IF Mach_Control.U.TJ_iMode=1 OR AV THEN//在自动状态下
CASE 	Sticker_Step2 OF
		0://判断备胶是否完成，贴胶冶具夹爪张开
				IF Mach_Control.TJ_b.StickPermit THEN//贴胶允许
						Sticker_Step2:=100;
				END_IF
		100:
				Mach_Control.TJ_b.StickPermit:=FALSE;//贴胶允许
				Mach_Control.TJ_b.StickFinish:=FALSE;//贴胶完成			
				Sticker_Step2:=200;
		200:
				IF NOT Sticker_SinStepMode THEN		
						IF 	Mach_Control.TJ_b.StickerStandbyDone  THEN//备胶完成,	
								Sticker_Step2:=250;						
						END_IF
				END_IF
		250: 
			IF arrCyCtrl[arrCyNo.ElectValveName.PastesGlueVacuum].Io.DOStatus1  
			AND arrCyCtrl[arrCyNo.ElectValveName.PastesGlueVacuum].Io.DIOnSwitch THEN
				Sticker_Step2:=300;
			ELSE
				Mach_Control.TJ_b.StickerStandbyDone:=FALSE;
				Mach_Control.TJ_b.Error[11]:=TRUE;//叠台贴胶头贴胶时无贴胶报警
				Sticker_Step2:=200;	
			END_IF
		
		300:
		arrAxisCtrl[AxiseNo.AxisName.GluingRetracting].Cmd.fOverride:=100;
				IF Mach_Control.TJ_b.Sticking_L THEN//左短边贴胶
					Sticker_Step2:=400;		
				ELSIF  Mach_Control.TJ_b.Sticking_R THEN//右短边贴胶
					Sticker_Step2:=450;		
				ELSIF Mach_Control.TJ_b.Sticking_Lg THEN//非极耳侧长边贴胶
					Sticker_Step2:=500;	
				ELSIF Mach_Control.TJ_b.Sticking_Lg2  THEN//极耳侧长边贴胶
					Sticker_Step2:=550;				
				END_IF	
		400://贴胶头移动左短边贴胶位
				IF NOT Sticker_SinStepMode THEN		
							IF GluingRetractingagree 
									AND  arrAxisCtrl[AxiseNo.AxisName.GluingRetracting].Status.Homed 
									AND arrAxisCtrl[AxiseNo.AxisName.GluingRetracting].Status.NoMoving 
									AND arrCyCtrl[arrCyNo.CylinderName.GlueClampsCy].Status.OFFState THEN
									IF arrAxisCtrl[AxiseNo.AxisName.GluingRetracting].Cmd.arrbRealPoint[2] THEN
											Mach_Control.TJ_b.Sticking_L:=FALSE;//左短边贴胶
											arrAxisCtrl[AxiseNo.AxisName.GluingRetracting].Cmd.iGoSetPos:=0;
											arrCyCtrl[arrCyNo.ElectValveName.PastesGlueVacuum].Cmd.bOFF:=TRUE;//备胶贴胶头真空关
											IF Mach_Control.TJ_b.SinStepMode THEN//贴胶单眇模式
													Sticker_SinStepMode:=TRUE;
											ELSE
													Sticker_SinStepMode:=FALSE;
											END_IF																						
											Sticker_Step2:=600;
									ELSE
											arrAxisCtrl[AxiseNo.AxisName.GluingRetracting].Cmd.iGoSetPos:=2;//贴胶头前进到贴胶位
									END_IF
										
							END_IF
							IF LREAL_TO_REAL(arrAxisCtrl[AxiseNo.AxisName.GluingRetracting].Status.fActPos) >= (arrAxisPar[AxiseNo.AxisName.GluingRetracting].arrTargetPoint[2]-30) THEN
									arrAxisCtrl[AxiseNo.AxisName.GluingRetracting].Cmd.fOverride:=5;
							END_IF
				END_IF
		450://贴胶头移动右短边贴胶位
				IF NOT Sticker_SinStepMode THEN		
						IF GluingRetractingagree 
						AND arrAxisCtrl[AxiseNo.AxisName.GluingRetracting].Status.Homed 
						AND arrAxisCtrl[AxiseNo.AxisName.GluingRetracting].Status.NoMoving 
						AND arrCyCtrl[arrCyNo.CylinderName.GlueClampsCy].Status.OFFState THEN
								IF arrAxisCtrl[AxiseNo.AxisName.GluingRetracting].Cmd.arrbRealPoint[3] THEN
										Mach_Control.TJ_b.Sticking_R:=FALSE;//左短边贴胶
										arrAxisCtrl[AxiseNo.AxisName.GluingRetracting].Cmd.iGoSetPos:=0;							
										arrCyCtrl[arrCyNo.ElectValveName.PastesGlueVacuum].Cmd.bOFF:=TRUE;//备胶贴胶头真空关
										IF Mach_Control.TJ_b.SinStepMode THEN//贴胶单眇模式
												Sticker_SinStepMode:=TRUE;
										ELSE
												Sticker_SinStepMode:=FALSE;
										END_IF																						
										Sticker_Step2:=600;
								ELSE
										arrAxisCtrl[AxiseNo.AxisName.GluingRetracting].Cmd.iGoSetPos:=3;//贴胶头前进到贴胶位
								END_IF	
						END_IF	
							IF LREAL_TO_REAL(arrAxisCtrl[AxiseNo.AxisName.GluingRetracting].Status.fActPos) >= (arrAxisPar[AxiseNo.AxisName.GluingRetracting].arrTargetPoint[3]-30) THEN
									arrAxisCtrl[AxiseNo.AxisName.GluingRetracting].Cmd.fOverride:=5;
							END_IF							
				END_IF
		500://非极耳侧长边贴胶
				IF NOT Sticker_SinStepMode THEN		
					IF GluingRetractingagree 
					AND arrAxisCtrl[AxiseNo.AxisName.GluingRetracting].Status.Homed 
					AND arrAxisCtrl[AxiseNo.AxisName.GluingRetracting].Status.NoMoving 
					AND arrCyCtrl[arrCyNo.CylinderName.GlueClampsCy].Status.OFFState THEN
						IF arrAxisCtrl[AxiseNo.AxisName.GluingRetracting].Cmd.arrbRealPoint[4] THEN
								Mach_Control.TJ_b.Sticking_Lg:=FALSE;//非极耳侧长边贴胶
								arrAxisCtrl[AxiseNo.AxisName.GluingRetracting].Cmd.iGoSetPos:=0;							
								arrCyCtrl[arrCyNo.ElectValveName.PastesGlueVacuum].Cmd.bOFF:=TRUE;//备胶贴胶头真空关
								IF Mach_Control.TJ_b.SinStepMode THEN//贴胶单眇模式
										Sticker_SinStepMode:=TRUE;
								ELSE
										Sticker_SinStepMode:=FALSE;
								END_IF																						
								Sticker_Step2:=600;
						ELSE
								arrAxisCtrl[AxiseNo.AxisName.GluingRetracting].Cmd.iGoSetPos:=4;//贴胶头前进到贴长边位
						END_IF		
					END_IF	
							IF LREAL_TO_REAL(arrAxisCtrl[AxiseNo.AxisName.GluingRetracting].Status.fActPos) >= (arrAxisPar[AxiseNo.AxisName.GluingRetracting].arrTargetPoint[4]-30) THEN
									arrAxisCtrl[AxiseNo.AxisName.GluingRetracting].Cmd.fOverride:=5;
							END_IF
				END_IF
	
			550://极耳侧长边贴胶
				IF NOT Sticker_SinStepMode THEN		
					IF GluingRetractingagree 
					AND arrAxisCtrl[AxiseNo.AxisName.GluingRetracting].Status.Homed 
					AND arrAxisCtrl[AxiseNo.AxisName.GluingRetracting].Status.NoMoving 
					AND arrCyCtrl[arrCyNo.CylinderName.GlueClampsCy].Status.OFFState THEN
						IF arrAxisCtrl[AxiseNo.AxisName.GluingRetracting].Cmd.arrbRealPoint[5] THEN
								Mach_Control.TJ_b.Sticking_Lg2:=FALSE;//极耳侧长边贴胶
								arrAxisCtrl[AxiseNo.AxisName.GluingRetracting].Cmd.iGoSetPos:=0;							
								arrCyCtrl[arrCyNo.ElectValveName.PastesGlueVacuum].Cmd.bOFF:=TRUE;//备胶贴胶头真空关
								IF Mach_Control.TJ_b.SinStepMode THEN//贴胶单眇模式
										Sticker_SinStepMode:=TRUE;
								ELSE
										Sticker_SinStepMode:=FALSE;
								END_IF																						
								Sticker_Step2:=600;
						ELSE
								arrAxisCtrl[AxiseNo.AxisName.GluingRetracting].Cmd.iGoSetPos:=5;//贴胶头前进到贴长边位
						END_IF		
					END_IF	
							IF LREAL_TO_REAL(arrAxisCtrl[AxiseNo.AxisName.GluingRetracting].Status.fActPos) >= (arrAxisPar[AxiseNo.AxisName.GluingRetracting].arrTargetPoint[5]-30) THEN
									arrAxisCtrl[AxiseNo.AxisName.GluingRetracting].Cmd.fOverride:=5;
							END_IF
				END_IF
			
		600:	
				IF NOT Sticker_SinStepMode THEN	
						TON_Sticker[4].IN:=FALSE;
						arrCyCtrl[arrCyNo.CylinderName.GlueClampsCy].Cmd.bON:=TRUE;//贴胶夹爪气缸夹紧
						IF arrCyCtrl[arrCyNo.CylinderName.GlueClampsCy].Status.ONState AND NOT arrCyCtrl[arrCyNo.CylinderName.GlueClampsCy].Status.Error1 THEN
								IF Mach_Control.TJ_b.SinStepMode THEN//贴胶单眇模式
									Sticker_SinStepMode:=TRUE;
								ELSE
									Sticker_SinStepMode:=FALSE;
								END_IF		
						TON_Sticker[4].IN:=TRUE;
							IF TON_Sticker[4].Q THEN
								Sticker_Step2:=700;	
								TON_Sticker[4].IN:=FALSE;
							END_IF		
						END_IF
				END_IF
		700:				
				IF NOT Sticker_SinStepMode THEN	
						arrCyCtrl[arrCyNo.CylinderName.GlueClampsCy].Cmd.bOFF:=TRUE;//贴胶夹爪气缸松开
						IF arrCyCtrl[arrCyNo.CylinderName.GlueClampsCy].Status.OFFState AND NOT arrCyCtrl[arrCyNo.CylinderName.GlueClampsCy].Status.Error2 THEN
								IF Mach_Control.TJ_b.SinStepMode THEN//贴胶单眇模式
										Sticker_SinStepMode:=TRUE;
								ELSE
										Sticker_SinStepMode:=FALSE;
								END_IF	
								arrAxisCtrl[AxiseNo.AxisName.GluingRetracting].Cmd.fOverride:=100;		
								Sticker_Step2:=800;
						END_IF
				END_IF
		800:
					IF NOT Sticker_SinStepMode THEN		
							IF GluingRetractingagree AND  arrAxisCtrl[AxiseNo.AxisName.GluingRetracting].Status.Homed AND arrAxisCtrl[AxiseNo.AxisName.GluingRetracting].Status.NoMoving THEN
									IF arrAxisCtrl[AxiseNo.AxisName.GluingRetracting].Cmd.arrbRealPoint[1] THEN
											arrAxisCtrl[AxiseNo.AxisName.GluingRetracting].Cmd.iGoSetPos:=0;
											Mach_Control.TJ_b.StickerStandbyDone:=FALSE;//复位备胶完成
											Mach_Control.TJ_b.StickFinish :=TRUE;//贴胶完成	
											Mach_Control.TJ_b.StickPermit:=false;//贴胶允许复位	
											IF Mach_Control.TJ_b.SinStepMode THEN//贴胶单眇模式
													Sticker_SinStepMode:=TRUE;
											ELSE
													Sticker_SinStepMode:=FALSE;
											END_IF																						
											Sticker_Step2:=900;
									ELSE
										arrAxisCtrl[AxiseNo.AxisName.GluingRetracting].Cmd.iGoSetPos:=1;//贴胶头前进到初始位
									END_IF
							END_IF	
					END_IF
			900:
					Sticker_Step2:=0;	
END_CASE
END_IF


CASE Sticker_Step0 OF
			1100://贴胶完成，允许下电芯，等待下电芯夹紧完成				
				IF Mach_Control.TJ_b.StickerOffloadingDone THEN
					Mach_Control.TJ_b.StickerFlag:=FALSE;
					Mach_Control.TJ_b.StickerOffloadingDone:=FALSE;						
					Sticker_Step0:=1200;
				END_IF
END_CASE


IF Sticker_Step0=4600 THEN
	Mach_Control.TJ_b.Stick_Judge:=TRUE;
ELSIF Sticker_Step0=2100 AND Sticker_Step0=2600 AND Sticker_Step0=3100 AND Sticker_Step0=3600 THEN
	Mach_Control.TJ_b.Stick_Judge:=FALSE;
END_IF
END_ACTION

ACTION _02BlueGlue_Auto:

(*
//蓝胶检测自动
DT_BlueGlue(
	Enable:=Mach_Control.U.DT_iMode=1 , //启动条件
	BlueSenser:=Mach_Control.se.BlueGluetsensor , //蓝胶检测信号
	An_Quantited:=Mach_Control.An_b.An_Quantited, //正极已叠极片数
	An_QuantitSet:=Par.stDT_date.An_Quantity , //正极设置极片数
	Ca_Quantited:=Mach_Control.Ca_b.Ca_Quantited, //负极已叠极片数
	Ca_QuantitSet:=Par.stDT_date.Ca_Quantity ,//负极设定极片数 
	Distance:=Par.stDT_date.Distance , //蓝胶检测到压刀的距离
	BluWidth:=Par.stDT_date.BluWidth , //蓝胶宽度
	Width:=Par.stDT_date.Width , //压刀外边宽
	BluGlueNG:=Mach_Control.DT_b.BluGlueNG );//电当蓝胶NG输出
	
	

//蓝胶标记
P2M_BlueFlag(
	Bnt_Blueflag:=Mach_Control.DT_b.stBnt_Blueflag , //蓝胶标记启动信号
	FlagDone:=P2M_BlueFlag.FlagDone , //蓝胶标记完成
	AixsoActPos:=arrAxis[AxiseNo.AxisName.SEPTAunwinding].NcToPlc.ActPos , //放卷轴当前位置
	Diameter:=Mach_Control.DT_b.fWindDiameter , //放卷轴当前卷径
	SetLenght:=Par.stDT_date.stSetLenght,//接带点到叠台的距离 3800
	fYDLength :=par.stDT_date.Width,
	rBnt_BlueflagCaNum :=Mach_Control.Ca_b.Ca_Quantited   , //叠台压刀外边宽
	FlagPoisn=> , //蓝胶NG标记
	NumberPos:=stNumberPos,//前一片数据
	NumberPos1:=stNumberPos1,//当前片数据
	NumberPos2:=stNumberPos2,
	rBnt_BlueflagNum :=DT_Ca_Quantited ,
	rBnt_Blueflaging:=Bnt_Blueflaging );//
	P2M_BlueFlag.FlagPoisn;	
	//
BulebntR_TRIG(CLK:=Mach_Control.DT_b.stBnt_Blueflag AND Mach_Control.DT_b.DT_Blue_TF   (*OR Mach_Control.btn.PoleInflationbtn*) , Q=> );
IF BulebntR_TRIG.Q THEN
	Bnt_Blueflaging:=TRUE;
	IF  (Par.stDT_date.An_Quantity+Par.stDT_date.Ca_Quantity-Mach_Control.An_b.An_Quantited-Mach_Control.Ca_b.Ca_Quantited)>=40 THEN
		Blueflaging:=TRUE;
	END_IF
END_IF	
*)
END_ACTION

ACTION _02Sticker_Auto:

TON_Sticker[0](PT:=T#0.2S);//拉胶气缸取胶延时
TON_Sticker[1](PT:=T#10S);//扫码超时报警延时
TON_Sticker[2](PT:=T#0.2S);//扫码超时报警延时
TON_Sticker[3](PT:=T#300MS);//扫码超时报警延时

IF Mach_Control.U.TJ_iMode<>1  THEN
				//一键备二维码胶
				rStickerStandbyCode_btn(CLK:=Mach_Control.btn.codeGluebtn , Q=> );
				fStickerStandbyCode_btn(CLK:=Mach_Control.btn.codeGluebtn , Q=> );
				IF rStickerStandbyCode_btn.Q THEN
					Mach_Control.TJ_b.StickerStandbyDone :=FALSE;
				END_IF
				IF fStickerStandbyCode_btn.Q THEN
					StandbyBule_Start:=FALSE;
					StandbyCode_Start:=TRUE;
				END_IF
				//一键备蓝胶
				rStickerStandbyBule_btn(CLK:=Mach_Control.btn.BlueGluebtn , Q=> );
				fStickerStandbyBule_btn(CLK:=Mach_Control.btn.BlueGluebtn , Q=> );
				IF rStickerStandbyBule_btn.Q THEN
					Mach_Control.TJ_b.StickerStandbyDone :=FALSE;
				END_IF
				IF fStickerStandbyBule_btn.Q THEN
					StandbyCode_Start:=FALSE;
					StandbyBule_Start:=TRUE;
				END_IF
END_IF

IF  StandbyBule_Start  THEN		
		Mach_Control.TJ_b.StickerStandbyBule:=FALSE;
END_IF

(*
//判断需要备什么胶,当设置的贴胶屏蔽时，置位已贴胶标记
IF Mach_Control.U.TJ_iMode=1 OR AV   THEN
			IF  NOT Mach_Control.TJ_b.StickerDoneNo[1]  AND NOT Mach_Control.TJ_b.Stickersetting[0]  THEN
				Mach_Control.TJ_b.StickerStandbyBule:=FALSE;//蓝胶备胶
				Mach_Control.TJ_b.StickerStandbyCode:=TRUE;//二维码备胶
				StandbyCode_Start:=FALSE;
				StandbyBule_Start:=FALSE;
			ELSIF (NOT Mach_Control.TJ_b.StickerDoneNo[2]  AND NOT Mach_Control.TJ_b.Stickersetting[1]) OR 
					(NOT Mach_Control.TJ_b.StickerDoneNo[3]  AND NOT Mach_Control.TJ_b.Stickersetting[2]) OR 
					(NOT Mach_Control.TJ_b.StickerDoneNo[4]  AND NOT Mach_Control.TJ_b.Stickersetting[3]) OR 
					(NOT Mach_Control.TJ_b.StickerDoneNo[5]  AND NOT Mach_Control.TJ_b.Stickersetting[4]) OR 
					(NOT Mach_Control.TJ_b.StickerDoneNo[6]  AND NOT Mach_Control.TJ_b.Stickersetting[5]) OR 
					(NOT Mach_Control.TJ_b.StickerDoneNo[7]  AND NOT Mach_Control.TJ_b.Stickersetting[6]) THEN
				Mach_Control.TJ_b.StickerStandbyBule:=TRUE;//蓝胶备胶
				Mach_Control.TJ_b.StickerStandbyCode:=FALSE;//二维码备胶	
				StandbyCode_Start:=FALSE;
				StandbyBule_Start:=FALSE;		
			END_IF
END_IF
*)


GluingUpDownPoint1:=ABS(arrAxisPar[AxiseNo.AxisName.GluingUpDown].arrTargetPoint[1]-arrAxisPar[AxiseNo.AxisName.GluingUpDown].arrTargetPoint[2]);
GluingUpDownPoint3:=ABS(GluingUpDownPoint2-arrAxisPar[AxiseNo.AxisName.GluingUpDown].arrTargetPoint[1]);
IF GluingUpDownPoint3-GluingUpDownPoint1>=2 THEN
	GluingUpDownPoint4:=2;
ELSIF GluingUpDownPoint3-GluingUpDownPoint1<=-2 THEN
	GluingUpDownPoint4:=-2;
ELSE
	GluingUpDownPoint4:=GluingUpDownPoint3-GluingUpDownPoint1;
END_IF

rMarkesensorR_TRIG(CLK:=Mach_Control.se.Markesensor , Q=> );

IF (Mach_Control.U.TJ_iMode=1 OR StandbyCode_Start OR StandbyBule_Start OR AV) AND NOT TJ_Error THEN//在自动状态下
	
//贴胶备胶自动
	
CASE Sticker_Step1 OF
		0://判断贴胶备胶是否完成
				IF NOT Sticker_SinStepMode THEN
						IF NOT Mach_Control.TJ_b.StickerStandbyDone THEN//备胶没有完成，贴胶头前进后退轴在安全位
								IF Mach_Control.TJ_b.SinStepMode THEN//贴胶单眇模式
									Sticker_SinStepMode:=TRUE;
								ELSE
									Sticker_SinStepMode:=FALSE;
								END_IF
								Sticker_Step1:=10;					
						END_IF
				END_IF
		10://备二维码胶真空1、备蓝胶真空1	
				//arrCyCtrl[arrCyNo.ElectValveName.codeGlueVacuum1].Cmd.bON:=TRUE;//备二维码胶真空1						
				arrCyCtrl[arrCyNo.ElectValveName.BlueGlueVacuum1].Cmd.bON:=TRUE;//备蓝胶真空1					
				Sticker_Step1:=20;			
		20://贴胶台具气缸张开、贴胶头前进轴回初始位
				IF NOT Sticker_SinStepMode THEN
						IF(GluingRetractingagree OR  arrAxisCtrl[AxiseNo.AxisName.GluingRetracting].Cmd.arrbRealPoint[1])AND
							arrAxisCtrl[AxiseNo.AxisName.GluingRetracting].Status.Homed AND arrAxisCtrl[AxiseNo.AxisName.GluingRetracting].Status.NoMoving THEN
								IF arrAxisCtrl[AxiseNo.AxisName.GluingRetracting].Cmd.arrbRealPoint[1] THEN
										arrAxisCtrl[AxiseNo.AxisName.GluingRetracting].Cmd.iGoSetPos:=0;						
										IF Mach_Control.TJ_b.SinStepMode THEN//贴胶单眇模式
												Sticker_SinStepMode:=TRUE;
										ELSE
												Sticker_SinStepMode:=FALSE;
										END_IF
										Sticker_Step1:=30;
								ELSE
										arrAxisCtrl[AxiseNo.AxisName.GluingRetracting].Cmd.iGoSetPos:=1;//贴胶头前进到贴胶位
								END_IF
						END_IF
				END_IF					
	   30://贴胶压胶气缸伸出，备胶气缸伸出
				IF NOT Sticker_SinStepMode THEN  
						arrCyCtrl[arrCyNo.CylinderName.GluePressCy].Cmd.bON:=TRUE;//贴胶压胶气缸伸出
						arrCyCtrl[arrCyNo.CylinderName.CodeGluePressCy].Cmd.bON:=TRUE;//贴胶压二维码胶气缸伸出
						IF arrCyCtrl[arrCyNo.CylinderName.CodeGluePressCy].Io.DIOnSwitch THEN
								arrCyCtrl[arrCyNo.CylinderName.CodeStandbyGlueCy].Cmd.bON:=TRUE;//贴胶备二维码胶气缸伸出
						END_IF
						IF Mach_Control.TJ_b.SinStepMode THEN//贴胶单眇模式
								Sticker_SinStepMode:=TRUE;
						ELSE
								Sticker_SinStepMode:=FALSE;
						END_IF
						IF arrCyCtrl[arrCyNo.CylinderName.GluePressCy].Status.ONState AND arrCyCtrl[arrCyNo.CylinderName.CodeGluePressCy].Status.ONState THEN
								Sticker_Step1:=40;	
						END_IF
				END_IF
		40://判断贴蓝胶、二维码胶
				IF NOT Sticker_SinStepMode THEN
					//IF Mach_Control.TJ_b.StickerStandbyBule OR StandbyBule_Start THEN//备蓝胶请求
					IF Mach_Control.TJ_b.SinStepMode THEN//贴胶单眇模式
							Sticker_SinStepMode:=TRUE;
					ELSE
							Sticker_SinStepMode:=FALSE;
					END_IF								
					arrCyCtrl[arrCyNo.CylinderName.StandbyGlueCy].Cmd.bON:=TRUE;//备蓝胶气缸伸出
					IF 	arrCyCtrl[arrCyNo.CylinderName.StandbyGlueCy].Io.DIOnSwitch THEN
							Sticker_Step1:=200;
					END_IF
					//END_IF	
				END_IF			
		200:// 二维码胶、蓝胶切胶气缸伸出，拉胶气缸伸出，拉胶升降轴移至拉蓝胶起始位
				IF NOT Sticker_SinStepMode THEN			
						arrCyCtrl[arrCyNo.CylinderName.codeGlueCutCy].Cmd.bON:=TRUE;//贴胶切二维码胶气缸伸出
						arrCyCtrl[arrCyNo.CylinderName.GlueCutCy].Cmd.bON:=TRUE;//贴胶切胶气缸伸出
						arrCyCtrl[arrCyNo.CylinderName.PullGlueCy].Cmd.bON:=TRUE;//拉胶气缸伸出
						arrCyCtrl[arrCyNo.CylinderName.StandbyGlueCy].Cmd.bOFF:=TRUE;//备蓝胶气缸伸出
						IF  GluingUpDownagree AND arrAxisCtrl[AxiseNo.AxisName.GluingUpDown].Status.Homed AND arrAxisCtrl[AxiseNo.AxisName.GluingUpDown].Status.NoMoving THEN
								IF arrAxisCtrl[AxiseNo.AxisName.GluingUpDown].Cmd.arrbRealPoint[9] THEN
										arrAxisCtrl[AxiseNo.AxisName.GluingUpDown].Cmd.iGoSetPos:=0;
										IF Mach_Control.TJ_b.SinStepMode THEN//贴胶单眇模式
												Sticker_SinStepMode:=TRUE;
										ELSE
												Sticker_SinStepMode:=FALSE;
										END_IF
										Sticker_Step1:=205;	
								ELSE
										arrAxisCtrl[AxiseNo.AxisName.GluingUpDown].Cmd.iGoSetPos:=9;//拉胶升降轴至拉蓝胶起始位
								END_IF
						END_IF		
				END_IF
		205:
				IF NOT Sticker_SinStepMode THEN
						IF  GluingUpDownagree AND arrAxisCtrl[AxiseNo.AxisName.GluingUpDown].Status.Homed AND arrAxisCtrl[AxiseNo.AxisName.GluingUpDown].Status.NoMoving THEN
								IF arrAxisCtrl[AxiseNo.AxisName.GluingUpDown].Cmd.arrbRealPoint[3] THEN
										arrAxisCtrl[AxiseNo.AxisName.GluingUpDown].Cmd.iGoSetPos:=0;
										IF Mach_Control.TJ_b.SinStepMode THEN//贴胶单眇模式
												Sticker_SinStepMode:=TRUE;
										ELSE
												Sticker_SinStepMode:=FALSE;
										END_IF
										Sticker_Step1:=210;	
								ELSE
										arrAxisCtrl[AxiseNo.AxisName.GluingUpDown].Cmd.iGoSetPos:=3;//拉胶升降轴至拉蓝胶起始位
								END_IF
						END_IF		
				END_IF
			210://拉胶升降气缸收回,取胶
				IF NOT Sticker_SinStepMode THEN			
						arrCyCtrl[arrCyNo.CylinderName.PullGlueCy].Cmd.bOFF:=TRUE;//拉胶气缸收回	
						arrCyCtrl[arrCyNo.CylinderName.GluePressCy].Cmd.bOFF:=TRUE;//贴胶压胶气缸伸出
						arrCyCtrl[arrCyNo.CylinderName.PullGluePoleCy].Cmd.bOFF:=TRUE;//拉胶抱紧气缸松开
						IF arrCyCtrl[arrCyNo.CylinderName.PullGlueCy].Io.DIOFFSwitch THEN
								IF NOT TON_Sticker[0].Q THEN
										TON_Sticker[0].IN:=TRUE;
								ELSE
										TON_Sticker[0].IN:=FALSE;
										IF Mach_Control.TJ_b.SinStepMode THEN//贴胶单眇模式
												Sticker_SinStepMode:=TRUE;
										ELSE
												Sticker_SinStepMode:=FALSE;
										END_IF
								Sticker_Step1:=220;
								END_IF
						END_IF	
				END_IF
		220://取胶滚胶位
				IF NOT Sticker_SinStepMode THEN			
						arrCyCtrl[arrCyNo.CylinderName.PullGluePoleCy].Cmd.bOFF:=TRUE;//拉胶抱紧气缸松开
						IF   arrAxisCtrl[AxiseNo.AxisName.GluingUpDown].Status.Homed AND arrAxisCtrl[AxiseNo.AxisName.GluingUpDown].Status.NoMoving THEN
								IF arrAxisCtrl[AxiseNo.AxisName.GluingUpDown].Cmd.arrbRealPoint[7] THEN
										arrAxisCtrl[AxiseNo.AxisName.GluingUpDown].Cmd.iGoSetPos:=0;
										IF Mach_Control.TJ_b.SinStepMode THEN//贴胶单眇模式
												Sticker_SinStepMode:=TRUE;
										ELSE
												Sticker_SinStepMode:=FALSE;
										END_IF
										Sticker_Step1:=221;	
								ELSE
										arrAxisCtrl[AxiseNo.AxisName.GluingUpDown].Cmd.iGoSetPos:=7;//拉胶升降轴取胶滚胶位
								END_IF
						END_IF
				END_IF	
		221://
				IF NOT Sticker_SinStepMode THEN
						IF NOT TON_Sticker[0].Q THEN
								arrCyCtrl[arrCyNo.ElectValveName.BlueGlueVacuum1].Cmd.bOFF:=TRUE;//备蓝胶真空1关
								arrCyCtrl[arrCyNo.ElectValveName.codeGlueVacuum2].Cmd.bOFF:=TRUE;//备二维码胶真空2关
								arrCyCtrl[arrCyNo.ElectValveName.PastesGlueVacuum].Cmd.bOFF:=TRUE;//备胶贴胶头真空关
								arrCyCtrl[arrCyNo.CylinderName.PullGluePoleCy].Cmd.bON:=TRUE;//拉胶抱紧气缸抱紧
								TON_Sticker[0].IN:=TRUE;
						ELSE
								TON_Sticker[0].IN:=FALSE;
								IF Mach_Control.TJ_b.SinStepMode THEN//贴胶单眇模式
										Sticker_SinStepMode:=TRUE;
								ELSE
										Sticker_SinStepMode:=FALSE;
								END_IF								
								Sticker_Step1:=230;	;	
						END_IF
				END_IF
		230://拉胶升降气缸伸出，拉胶升降气缸移动至拉蓝胶终点位
				IF NOT Sticker_SinStepMode THEN			
						arrCyCtrl[arrCyNo.CylinderName.codeGlueCutCy].Cmd.bON:=TRUE;//贴胶切二维码胶气缸伸出
						arrCyCtrl[arrCyNo.CylinderName.GlueCutCy].Cmd.bON:=TRUE;//贴胶切胶气缸伸出
						arrCyCtrl[arrCyNo.CylinderName.PullGlueCy].Cmd.bON:=TRUE;//拉胶气缸伸出
						arrCyCtrl[arrCyNo.CylinderName.PullGluePoleCy].Cmd.bON:=TRUE;//拉胶抱紧气缸抱紧
						IF  GluingUpDownagree AND arrAxisCtrl[AxiseNo.AxisName.GluingUpDown].Status.Homed AND arrAxisCtrl[AxiseNo.AxisName.GluingUpDown].Status.NoMoving THEN
								IF arrAxisCtrl[AxiseNo.AxisName.GluingUpDown].Cmd.arrbRealPoint[4] THEN
										arrAxisCtrl[AxiseNo.AxisName.GluingUpDown].Cmd.iGoSetPos:=0;
										IF Mach_Control.TJ_b.SinStepMode THEN//贴胶单眇模式
												Sticker_SinStepMode:=TRUE;
										ELSE
												Sticker_SinStepMode:=FALSE;
										END_IF
										Sticker_Step1:=240;	
								ELSE
										arrAxisCtrl[AxiseNo.AxisName.GluingUpDown].Cmd.iGoSetPos:=4;//拉胶升降轴至拉蓝胶终点位
								END_IF
						END_IF
				END_IF					
		240://拉胶气缸收回
				IF NOT Sticker_SinStepMode THEN			
						arrCyCtrl[arrCyNo.CylinderName.PullGlueCy].Cmd.bOFF:=TRUE;//拉胶气缸收回		
						arrCyCtrl[arrCyNo.CylinderName.PullGluePoleCy].Cmd.bOFF:=TRUE;//拉胶抱紧气缸松开	
						arrCyCtrl[arrCyNo.ElectValveName.BlueGlueVacuum1].Cmd.bON:=TRUE;//备蓝胶真空1
						arrCyCtrl[arrCyNo.ElectValveName.BlueGlueVacuum2].Cmd.bON:=TRUE;//备蓝胶真空2	
						arrCyCtrl[arrCyNo.ElectValveName.codeGlueVacuum1].Cmd.bON:=TRUE;//备二维码胶真空1
						arrCyCtrl[arrCyNo.ElectValveName.codeGlueVacuum2].Cmd.bON:=TRUE;//备二维码胶真空2																			
						IF arrCyCtrl[arrCyNo.CylinderName.PullGlueCy].Status.OFFState THEN
								IF NOT TON_Sticker[0].Q THEN
										TON_Sticker[0].IN:=TRUE;
								ELSE
										TON_Sticker[0].IN:=FALSE;
										IF Mach_Control.TJ_b.SinStepMode THEN//贴胶单眇模式
												Sticker_SinStepMode:=TRUE;
										ELSE
												Sticker_SinStepMode:=FALSE;
										END_IF					
								Sticker_Step1:=250;
								END_IF
						END_IF	
				END_IF
		250:	//拉胶升降轴至切胶滚胶位	
				IF NOT Sticker_SinStepMode THEN			
						IF   arrAxisCtrl[AxiseNo.AxisName.GluingUpDown].Status.Homed AND arrAxisCtrl[AxiseNo.AxisName.GluingUpDown].Status.NoMoving THEN
								IF arrAxisCtrl[AxiseNo.AxisName.GluingUpDown].Cmd.arrbRealPoint[8] THEN
										arrAxisCtrl[AxiseNo.AxisName.GluingUpDown].Cmd.iGoSetPos:=0;
										IF Mach_Control.TJ_b.SinStepMode THEN//贴胶单眇模式
												Sticker_SinStepMode:=TRUE;
										ELSE
												Sticker_SinStepMode:=FALSE;
										END_IF
										Sticker_Step1:=255;	
								ELSE
										arrAxisCtrl[AxiseNo.AxisName.GluingUpDown].Cmd.iGoSetPos:=8;//拉胶升降轴至切胶滚胶位
								END_IF
						END_IF
				END_IF	
	
		255://20230205修改切胶动作
				arrCyCtrl[arrCyNo.CylinderName.GluePressCy].Cmd.bON:=TRUE;//贴胶压胶气缸伸出
				IF arrCyCtrl[arrCyNo.CylinderName.GluePressCy].Status.ONState THEN//贴胶压胶气缸伸出
						Sticker_Step1:=260;		
				END_IF
		
		260://切二维码胶气缸收回，切胶
				IF NOT Sticker_SinStepMode THEN	
						arrCyCtrl[arrCyNo.ElectValveName.PastesGlueVacuum].Cmd.bON:=TRUE;//备胶贴胶头真空		
						arrCyCtrl[arrCyNo.CylinderName.GlueCutCy].Cmd.bOFF:=TRUE;//切蓝胶气缸收回
						IF arrCyCtrl[arrCyNo.CylinderName.GlueCutCy].Status.OFFState THEN													
									IF Mach_Control.TJ_b.SinStepMode THEN//贴胶单眇模式
											Sticker_SinStepMode:=TRUE;
									ELSE
											Sticker_SinStepMode:=FALSE;
									END_IF															
									Sticker_Step1:=270;	
						END_IF	
				END_IF
		270://拉胶气缸伸出、切胶气缸伸出、拉胶升降轴回初始位
				IF NOT Sticker_SinStepMode THEN			
						arrCyCtrl[arrCyNo.CylinderName.codeGlueCutCy].Cmd.bON:=TRUE;//贴胶切二维码胶气缸伸出
						arrCyCtrl[arrCyNo.CylinderName.GlueCutCy].Cmd.bON:=TRUE;//贴胶切胶气缸伸出
						arrCyCtrl[arrCyNo.CylinderName.PullGlueCy].Cmd.bON:=TRUE;//拉胶气缸伸出
						arrCyCtrl[arrCyNo.ElectValveName.BlueGlueVacuum2].Cmd.bON:=FALSE;//备蓝胶真空2	
						arrCyCtrl[arrCyNo.ElectValveName.codeGlueVacuum2].Cmd.bON:=FALSE;//备二维码胶真空2
						arrCyCtrl[arrCyNo.ElectValveName.BlueGlueVacuum2].Cmd.bOFF:=TRUE;//备蓝胶真空2	
						arrCyCtrl[arrCyNo.ElectValveName.codeGlueVacuum2].Cmd.bOFF:=TRUE;//备二维码胶真空2								
						IF  GluingUpDownagree AND arrAxisCtrl[AxiseNo.AxisName.GluingUpDown].Status.Homed AND arrAxisCtrl[AxiseNo.AxisName.GluingUpDown].Status.NoMoving THEN
								IF arrAxisCtrl[AxiseNo.AxisName.GluingUpDown].Cmd.arrbRealPoint[9] THEN
										arrAxisCtrl[AxiseNo.AxisName.GluingUpDown].Cmd.iGoSetPos:=0;
										IF Mach_Control.TJ_b.SinStepMode THEN//贴胶单眇模式
												Sticker_SinStepMode:=TRUE;
										ELSE
												Sticker_SinStepMode:=FALSE;
										END_IF
										Mach_Control.TJ_b.StickerStandbyDone:=TRUE;
										StandbyBule_Start:=FALSE;
										arrCyCtrl[arrCyNo.CylinderName.StandbyGlueCy].Cmd.bON:=TRUE;//备蓝胶气缸伸出		
										Sticker_Step1:=0;	
								ELSE
										arrAxisCtrl[AxiseNo.AxisName.GluingUpDown].Cmd.iGoSetPos:=9;//拉胶升降轴至拉蓝胶起始位
								END_IF
						END_IF		
				END_IF						
END_CASE
END_IF


IF Mach_Control.TJ_b.Error[5] AND Sticker_Step1>=260 AND Sticker_Step1<=270 THEN
	Sticker_Step1:=0;
	Mach_Control.TJ_b.StickerStandbyDone:=FALSE;
END_IF
END_ACTION

ACTION _02Sticker_AutoSbu1_Scan:
(*
Scan_TON[1](PT:=T#3MS);
Scan_TON[2](PT:=T#3MS);
Scan_TON[3](PT:=T#3MS);
Scan_TON[4](PT:=T#100MS);


//二维码胶扫码		
	CASE Stick_Step0 OF
		10:
			Scan_TON[1].IN:=FALSE;
			Scan_TON[2].IN:=FALSE;
			Scan_TON[3].IN:=FALSE;
			Stick_Step0:=20;
			
		20:
			fbinit_tcp:=TRUE;
			Scan_TON[1].IN:=TRUE;
			IF Scan_TON[1].Q THEN
				fbinit_tcp:=FALSE;
				Scan_TON[1].IN:=FALSE;
				Stick_Step0:=30;
			END_IF

		30:
			fbComOpen:=TRUE;
			Scan_TON[2].IN:=TRUE;
			IF Scan_TON[2].Q THEN
				fbComOpen:=FALSE;
				Scan_TON[2].IN:=FALSE;
				Stick_Step0:=40;
			END_IF

		40:
			IF bCS_CodeTcp.bComOpenDone THEN
				Stick_Step0:=50;
			END_IF
		
		50:
			bCS_CodeTcp.bLON:=TRUE;
			Scan_TON[3].IN:=TRUE;
			IF Scan_TON[3].Q THEN
				bCS_CodeTcp.bLON:=FALSE;
				Scan_TON[3].IN:=FALSE;
				Stick_Step0:=60;
			END_IF
		60:
			Scan_TON[4].IN:=TRUE;
			IF 	Scan_TON[4].Q THEN
				Stick_Step0:=70;
				Scan_TON[4].IN:=FALSE;
			END_IF

		70:
			IF  bCS_CodeTcp.Code_State=1  THEN
				Mach_Control.TJ_b.strCode:=bCS_CodeTcp.strCode;
				Mach_Control.TJ_b.Scan_gross:=bCS_CodeTcp.Code_State;
				Stick_Step0:=80;
				Mach_Control.TJ_b.ScanStarte:=FALSE;
				
			 ELSIF bCS_CodeTcp.Code_State=2 THEN
				 Mach_Control.TJ_b.Scan_gross:=bCS_CodeTcp.Code_State;
				 Stick_Step0:=80;
				 Mach_Control.TJ_b.ScanStarte:=FALSE;
			 ELSIF bCS_CodeTcp.bCodeConError OR Mach_Control.TJ_b.Error[0] THEN
				Stick_Step0:=6666;
				Mach_Control.TJ_b.ScanStarte:=FALSE;
			END_IF

	END_CASE

(*IF Mach_Control.TJ_b.ScanOK AND NOT   Mach_Control.TJ_b.ScanNG THEN
					Mach_Control.TJ_b.ScanStatus[0]:=TRUE;//扫码位的胶琮扫码OK
					Mach_Control.TJ_b.ScanStarte:=FALSE;//二维码扫码启动	
					TON_Sticker[1].IN:=FALSE;
					Stick_Step0:=6666;
				ELSIF NOT Mach_Control.TJ_b.ScanOK AND Mach_Control.TJ_b.ScanNG  THEN
					Mach_Control.TJ_b.ScanStatus[0]:=FALSE;//扫码位的胶琮扫码NG
					Mach_Control.TJ_b.ScanStarte:=FALSE;//二维码扫码启动	
					TON_Sticker[1].IN:=FALSE;	
					Stick_Step0:=6666;	
				ELSE
						IF NOT TON_Sticker[1].Q THEN
							TON_Sticker[1].IN:=TRUE;
						ELSE
							TON_Sticker[1].IN:=FALSE;
							Mach_Control.TJ_b.Error[0]:=TRUE;//扫码超时报警
							Mach_Control.TJ_b.ScanStarte:=FALSE;//二维码扫码启动	
							Stick_Step0:=9999;	
						END_IF
				END_IF*)

	
	
		
			
					
(*
上升沿触发 fbComOpen,  bComOpenDone连接完成；
触发fbLON拍照；
*)
bCS_CodeTcp(
	bLON:=bCS_CodeTcp.bLON,                           	// 扫码触发
	sRemoteHost:=Par.Code.sRemoteHost	,					//后段扫码枪；sRemoteHost:='192.168.10.25'
	bComOpen:=fbComOpen,           //扫码Tcp 连接，上升沿；
	binit_tcp:=fbinit_tcp,					//初始化功能块，上升沿；
	bComOpenDone=>, 			 //扫码Tcp 打开OK
    bCodeConError =>Mach_Control.TJ_b.Error[0],            	//扫码通讯故障
	bDone=>,                        	 //扫码完成
    bCodeError=>Mach_Control.TJ_b.Error[0],                  //扫码故障	
    strCode =>,                      //条码结果
	Code_State=>,					//扫码结果 1：OK  2：NG
);

bCS_CodeTcp.bDone;//这个需外部复位；
bCS_CodeTcp.strCode;
bCS_CodeTcp.Code_State;
bCS_CodeTcp.bComOpenDone;

*)
END_ACTION

ACTION _02Sticker_AutoSbu2_NG:

//贴胶踢废胶程序
		CASE 	Stick_Step2  OF 
		100://踢废胶
					arrCyCtrl[arrCyNo.CylinderName.GlueNGCy].Cmd.bON:=TRUE;//踢废胶升降气缸伸出
					IF 	 arrCyCtrl[arrCyNo.CylinderName.GlueNGCy].Io.DIOnSwitch THEN
						IF arrAxisCtrl[AxiseNo.AxisName.GluingRetracting].Status.Homed AND arrAxisCtrl[AxiseNo.AxisName.GluingRetracting].Status.NoMoving THEN
							IF arrAxisCtrl[AxiseNo.AxisName.GluingRetracting].Cmd.arrbRealPoint[6] THEN
								arrAxisCtrl[AxiseNo.AxisName.GluingRetracting].Cmd.iGoSetPos:=0;
								Mach_Control.TJ_b.StickerStandbyDone:=FALSE;//复位备胶完成
								IF Mach_Control.TJ_b.SinStepMode THEN//贴胶单眇模式
									Sticker_SinStepMode:=TRUE;
								ELSE
									Sticker_SinStepMode:=FALSE;
								END_IF																						
								Stick_Step2:=200;
							ELSE
								arrAxisCtrl[AxiseNo.AxisName.GluingRetracting].Cmd.iGoSetPos:=6;//踢废胶位
							END_IF
						END_IF	
					END_IF	
		120://贴胶冶具夹爪夹紧
					IF NOT Sticker_SinStepMode THEN		
						arrCyCtrl[arrCyNo.CylinderName.PullGlueModelCy].Cmd.bON:=TRUE;//贴胶冶具夹爪夹紧
						IF arrCyCtrl[arrCyNo.CylinderName.PullGlueModelCy].Io.DIOnSwitch THEN
							IF Mach_Control.TJ_b.SinStepMode THEN//贴胶单眇模式
								Sticker_SinStepMode:=TRUE;
							ELSE
								Sticker_SinStepMode:=FALSE;
							END_IF								
							Stick_Step2:=130;
						END_IF
					END_IF	
		130://贴胶夹爪张开，贴胶尖退回到初始位
					IF NOT Sticker_SinStepMode THEN		
							arrCyCtrl[arrCyNo.CylinderName.PullGlueModelCy].Cmd.bOFF:=TRUE;//贴胶冶具夹爪张开
							IF 	Mach_Control.TJ_b.StickerStandbyDone THEN
								IF arrCyCtrl[arrCyNo.CylinderName.PullGlueModelCy].Io.DIOFFSwitch AND arrAxisCtrl[AxiseNo.AxisName.GluingRetracting].Status.Homed AND arrAxisCtrl[AxiseNo.AxisName.GluingRetracting].Status.NoMoving THEN
									IF arrAxisCtrl[AxiseNo.AxisName.GluingRetracting].Cmd.arrbRealPoint[1] THEN
										arrAxisCtrl[AxiseNo.AxisName.GluingRetracting].Cmd.iGoSetPos:=0;
										IF Mach_Control.TJ_b.SinStepMode THEN//贴胶单眇模式
											Sticker_SinStepMode:=TRUE;
										ELSE
											Sticker_SinStepMode:=FALSE;
										END_IF																						
										Stick_Step2:=140;
									ELSE
										arrAxisCtrl[AxiseNo.AxisName.GluingRetracting].Cmd.iGoSetPos:=1;//贴胶头前进到备胶位
									END_IF
								END_IF						
						END_IF
					END_IF	
		140://踢废胶升降气缸纠回	
					arrCyCtrl[arrCyNo.CylinderName.GlueNGCy].Cmd.bOFF:=TRUE;//踢废胶升降气缸纠回
					IF 	arrCyCtrl[arrCyNo.CylinderName.GlueNGCy].Io	.DIOFFSwitch	THEN
						Stick_Step2:=6666;
					END_IF
		END_CASE
END_ACTION

ACTION _03Rectifydev_Auto:

//隔膜纠偏自动
IF Mach_Control.DT_b.RectifydevStarte OR Mach_Control.U.DT_iMode=1 OR (TailCurlStep3>=150 AND TailCurlStep3<=160  AND  Mach_Control.U.WJ_iMode=1 ) THEN
	 fbRectifyGM.Execute:=TRUE;
ELSE
	fbRectifyGM.Execute:=FALSE;
END_IF
//隔膜纠偏条件
(*
//fbRectifyGM.bRecEn:= arrAxis[AxiseNo.VirAxisName.VirGM].NcToPlc.SetVelo>=0.5 AND  ABS( arrAxis[AxiseNo.AxisName.SEPTATLine].NcToPlc.ActPos  )>=24 ;    //隔膜正向运动且隔膜包角OK位置 
fbRectifyGM.bRecEn:=((( 
                                    (LREAL_TO_REAL(arrAxisCtrl[AxiseNo.AxisName.SEPTATLine].Status.fActPos)>arrAxisPar[AxiseNo.AxisName.SEPTATLine].arrTargetPoint[1]+1    AND   
                                     LREAL_TO_REAL(arrAxisCtrl[AxiseNo.AxisName.SEPTATLine].Status.fActPos)<arrAxisPar[AxiseNo.AxisName.SEPTATLine].arrTargetPoint[1]+120) OR
                                    (LREAL_TO_REAL(arrAxisCtrl[AxiseNo.AxisName.SEPTATLine].Status.fActPos)<arrAxisPar[AxiseNo.AxisName.SEPTATLine].arrTargetPoint[2]-1    AND   
                                     LREAL_TO_REAL(arrAxisCtrl[AxiseNo.AxisName.SEPTATLine].Status.fActPos)>arrAxisPar[AxiseNo.AxisName.SEPTATLine].arrTargetPoint[2]-110) OR
									(TailCurlStep3>=1070 AND TailCurlStep3<=1080 AND  Mach_Control.U.WJ_iMode=1)                                                           OR 
                                    (TailCurlStep3>=150 AND TailCurlStep3<=160 AND  Mach_Control.U.WJ_iMode=1) AND Par.stDT_date.iRectifyMode=2))(* OR
									 (arrAxis[AxiseNo.VirAxisName.VirGM].NcToPlc.SetVelo>=5 AND  ABS( arrAxis[AxiseNo.AxisName.SEPTATLine].NcToPlc.ActPos  )>=24)  AND Par.stDT_date.iRectifyMode=1) *) OR Mach_Control.DT_b.RectifydevStarte) AND 
									 NOT Mach_Control.DT_b.RectifydevModel   ; //隔膜正向运动且隔膜包角OK位置 
*)

//纠偏条件		
(*							 
bRectifyRule[1]:=arrAxisCtrl[AxiseNo.AxisName.SEPTATLine].Status.fActPos>(arrAxisPar[AxiseNo.AxisName.SEPTATLine].arrTargetPoint[1]+5)    AND   
                                     arrAxisCtrl[AxiseNo.AxisName.SEPTATLine].Status.fSetPos<(arrAxisPar[AxiseNo.AxisName.SEPTATLine].arrTargetPoint[1]+Par.stDT_date.iRectifyAnPos);	//隔膜纠偏条件										 
									 
bRectifyRule[2]:=arrAxisCtrl[AxiseNo.AxisName.SEPTATLine].Status.fActPos<(arrAxisPar[AxiseNo.AxisName.SEPTATLine].arrTargetPoint[2]-5 )   AND   
                                     arrAxisCtrl[AxiseNo.AxisName.SEPTATLine].Status.fSetPos>(arrAxisPar[AxiseNo.AxisName.SEPTATLine].arrTargetPoint[2]-Par.stDT_date.iRectifyCaPos);
*)
								 
bRectifyRule[1]:=fbCamInGMDanserMove.iTableSel=2  AND   arrAxis[AxiseNo.AxisName.SEPTATLine].Status.Moving AND
                             arrAxisCtrl[AxiseNo.AxisName.SEPTATLine].Status.fSetPos<(arrAxisPar[AxiseNo.AxisName.SEPTATLine].arrTargetPoint[1]+Par.stDT_date.iRectifyAnPos);	//隔膜纠偏条件										 
									 
bRectifyRule[2]:=fbCamInGMDanserMove.iTableSel=1  AND   arrAxis[AxiseNo.AxisName.SEPTATLine].Status.Moving AND
                             arrAxisCtrl[AxiseNo.AxisName.SEPTATLine].Status.fSetPos>(arrAxisPar[AxiseNo.AxisName.SEPTATLine].arrTargetPoint[2]-Par.stDT_date.iRectifyCaPos);	
								 
bRectifyRule[3]:=TailCurlStep3>=1070 AND TailCurlStep3<=1080 AND  Mach_Control.U.WJ_iMode=1;		
bRectifyRule[4]:=TailCurlStep3>=150 AND TailCurlStep3<=160 AND  Mach_Control.U.WJ_iMode=1 AND Par.stDT_date.iRectifyMode=2;			
				 
fbRectifyGM.bRecEn:=NOT Mach_Control.DT_b.RectifydevModel AND( bRectifyRule[1] OR bRectifyRule[2] OR bRectifyRule[3] OR bRectifyRule[4] OR An_OverNGStep=1840 OR Ca_OverNGStep=1840)
                (*AND (Mach_Control.Ca_b.Ca_Quantited<5 OR Mach_Control.Ca_b.Ca_Quantited>9*) ; 


(*				 
IF (TailCurlStep3>=150 AND TailCurlStep3<=160) OR (TailCurlStep3>=1070 AND TailCurlStep3<=1080) THEN				  				 
		fRectifyTimeAdjust1:= Par.stDT_date.fRectifyTimeAdjust ;							 							 
ELSE								 
		fRectifyTimeAdjust1:= SEL( Mach_Control.An_b.An_Quantited>=1 AND Mach_Control.Ca_b.Ca_Quantited <Par.stDT_date.Ca_Quantity AND NOT  An_OverNGMark AND NOT Ca_OverNGMark  ,5   ,Par.stDT_date.DP_fRectifyTimeAdjust )               ;								 
END_IF 								 
*)
(*
IF  Mach_Control.An_b.An_Quantited<3 OR 
	 ((An_OverNGStep>1000 OR Ca_OverNGStep>1000 )(*AND  arrAxis[AxiseNo.VirAxisName.VirMain].Status.NotMoving	*)) OR 
	 (Mach_Control.Ca_b.Ca_Quantited= Par.stDT_date.Ca_Quantity  AND Mach_Control.An_b.An_Quantited= Par.stDT_date.An_Quantity)  THEN
	fRectifyTimeAdjust1:=3 ;	
ELSIF  Mach_Control.An_b.An_Quantited<4 THEN
	fRectifyTimeAdjust1:=Par.stDT_date.DP_fRectifyTimeAdjust+0.5 ;
ELSIF	(TailCurlStep3>=150 AND TailCurlStep3<=160) OR (TailCurlStep3>=1070 AND TailCurlStep3<=1080) THEN
	fRectifyTimeAdjust1:= Par.stDT_date.fRectifyTimeAdjust ;	
ELSE
	fRectifyTimeAdjust1:= Par.stDT_date.DP_fRectifyTimeAdjust ;	
END_IF									 
*)

IF (TailCurlStep3>=150 AND TailCurlStep3<=160) OR (TailCurlStep3>=1070 AND TailCurlStep3<=1080) THEN
   fRectifyTimeAdjust1:= Par.stDT_date.fRectifyTimeAdjust ;	
ELSE
	fRectifyTimeAdjust1:= Par.stDT_date.DP_fRectifyTimeAdjust ;	
END_IF										 
(*
IF Mach_Control.An_b.An_Quantited=4 AND Mach_Control.Ca_b.Ca_Quantited<>9 THEN
  fbRectifyGM.fSensorBalanceValue:=Par.stDT_date.fRectifyBalanceValue+0.7;
ELSE
  fbRectifyGM.fSensorBalanceValue:=Par.stDT_date.fRectifyBalanceValue;	
END_IF
*)									 
fbRectifyGM(
	bReset:=                      stSysState.bReset  ,  
	Execute:=                    fbRectifyGM.Execute  , 
	bCcw:=                       TRUE,//Mach_Control.DT_b.CWW , //纠偏方向选择
	iRectifyMode:=            Par.stDT_date.iRectifyMode , 
	bRecEn:=                   ,                         //纠偏容许条件
	fSensorActValue:=        Mach_Control.DT_b.RecDevPV , 
	fSensorActValue1:=       Mach_Control.DT_b.RecDevPV1 , 
	fSensorMaxValue:=       Par.stDT_date.fRectifyMaxValue , //从轴纠偏行程上限
	fSensorMinValue:=       Par.stDT_date.fRectifyMinValue , //从轴纠偏行程下限
	fSensorBalanceValue:=  Par.stDT_date.fRectifyBalanceValue,//纠偏平衡位置
	fTolerance:=                 Par.stDT_date.fRectifyfTolerance ,  //纠偏死区                        , 
	fGMLengthSet:=            Par.stDT_date.fRectifyGMLengthSet, //纠偏距离标定
	fTimeAdjust:=                fRectifyTimeAdjust1 , //纠偏时间标定
	bReady=> , 
	bAutoRunning=> , 
	Error=> , 
	Axis_Rectify1:=         arrAxis[AxiseNo.AxisName.SEPTAdeviation2] ,    
    Axis_Rectify2:=         arrAxis[AxiseNo.AxisName.SEPTAdeviation1] ,     
	//Axis_VirGM:=        arrAxis[AxiseNo.VirAxisName.VirGM] ,    
	Axis_Time:=          arrAxis[AxiseNo.VirAxisName.VirGM] ,     );   //arrAxis[AxiseNo.VirAxisName.VirTimeWind]

fbRectifyGM.bReady;
fbRectifyGM.bAutoRunning;//纠偏运行中
Mach_Control.DT_b.Error[21]:=fbRectifyGM.Error;//隔膜纠偏报警


//左右方向运动用同一个凸轮  
(*
IF  fbCamInVirGM.iTableSel=1 THEN
  fbCamInVirGM.ParCamIn.MasterScaling:=ABS(arrAxisPar[AxiseNo.AxisName.SEPTATLine] .arrTargetPoint[1]-arrAxisPar[AxiseNo.AxisName.SEPTATLine] .arrTargetPoint[2])/3600;
ELSIF  fbCamInVirGM.iTableSel=2 THEN
 fbCamInVirGM.ParCamIn.MasterScaling:=-ABS(arrAxisPar[AxiseNo.AxisName.SEPTATLine] .arrTargetPoint[1]-arrAxisPar[AxiseNo.AxisName.SEPTATLine] .arrTargetPoint[2])/3600;
END_IF
*)

(*
IF  fbCamInVirGM.iTableSel=1 THEN
  fbCamInVirGM.ParCamIn.MasterScaling:= (fMaxPos-fMinPos)/3600;
ELSIF  fbCamInVirGM.iTableSel=2 THEN
 fbCamInVirGM.ParCamIn.MasterScaling:=- (fMaxPos-fMinPos)/3600;
END_IF


fbCamInVirGM(
	Reset:=                      stSysState.bReset  , 
	bCamInExecute:=       fbCamInVirGM.bCamInExecute, 
	iTable1:=                   TableNo.M_GMLengthCalculate_L, 
	iTable2:=                    TableNo.M_GMLengthCalculate_L, 
	iTableSel:=               fbCamInVirGM.iTableSel , 
	ParCamIn:=                , 
  	axisMaster:=            arrAxis[AxiseNo.AxisName.SEPTATLine] ,  //AxiseNo.VirAxisName.VirMain   
	axisSlave:=               arrAxis[AxiseNo.VirAxisName.VirGM] ,  // arrAxis[AxiseNo.VirAxisName.VirGM]
	bError=> , 
	bReady=> , 
	bInSync=> );

fbCamInVirGM.bError;
fbCamInVirGM.bReady;
fbCamInVirGM.bInSync;
*)


rDtUse[5](CLK:=Mach_Control.DT_b.bRecDevBtn);//隔膜检测传感器标定按钮

//隔膜打皱报警------通过判断两个传感器偏差量大小分辨
IF rDtUse[5].Q THEN
	Par.stDT_date.rRecDev:=ABS(Mach_Control.DT_b.RecDevPV-Mach_Control.DT_b.RecDevPV1);//作为基准
END_IF

IF  Mach_Control.DT_b.bTensionOK AND Mach_Control.Ca_b.Ca_Quantited>=10  AND fbRectifyGM.bRecEn THEN//张力OK	&	 已叠层数超过N层	&	纠偏允许，开始判断
	IF ABS(ABS(Mach_Control.DT_b.RecDevPV-Mach_Control.DT_b.RecDevPV1)-Par.stDT_date.rRecDev)>=Par.stDT_date.rRecDevScope THEN
		Mach_Control.DT_b.Error_tips[3]:=TRUE;//隔膜打皱
	END_IF
END_IF

Rectifydev1:=Mach_Control.DT_b.RecDevPV-Par.stDT_date.fRectifyBalanceValue;//传感器1相当于基准值的变化
Rectifydev2:=Mach_Control.DT_b.RecDevPV1-Par.stDT_date.fRectifyBalanceValue;//传感器2相当于基准值的变化
//隔膜虚轴凸轮表
(*
fbCamInVirGM(
	Reset:=                     stSysState.bReset  , 
	bCamInExecute:=      fbCamInVirGM.bCamInExecute, 
	iTableSel:=                fbCamInVirGM.iTableSel, 
	bCreatTable:=          fbCamInVirGM.bCreatTable  ,           
	iTable:=                 TableNo.M_GMVir_L , 
    arrGMVirTableData:=     arrDeltaGMLengthAbs_L   , 
	axisSlave:=            arrAxis[AxiseNo.VirAxisName.VirGM] ,  
	axisMaster:=         arrAxis[AxiseNo.AxisName.SEPTATLine] ,  
	bCreatTableDone=> , 
	bCreatTableError=> , 
	bError=> , 
	bReady=> , 
	bInSync=> );
fbCamInVirGM.bCreatTableDone;
fbCamInVirGM.bCreatTableError;
fbCamInVirGM.bReady;
fbCamInVirGM.bError;
fbCamInVirGM.bInSync;



//尾卷平移与隔膜虚轴齿轮耦合
fbGearInGMvir(
	Reset:=            stSysState.bReset  , 
	fratio1:=           1, 
	bError=> , 
	bReady=> , 
	InGear=> , 
	bEnable:=  fbGearInGMvirbEnable , 
	master:=  arrAxis[AxiseNo.AxisName.TailCurlLine], 
	slave1:=    arrAxis[AxiseNo.VirAxisName.VirGM] );

fbGearInGMvir.bError;
fbGearInGMvir.bReady;
fbGearInGMvir.InGear;

*)

















(*
//隔膜纠偏自动
Rectifydev_V1(
	Enable:=Rectifydev_V1.Enable, //自动启动
	RestHMI:= Sys_Control.btn.System_Rrestbtn, //报警复位
	MasterNo:=AxiseNo.VirAxisName.VirTailCurl , //主轴号,时间主轴
	SlaveNo1:=AxiseNo.AxisName.SEPTAdeviation1 , //从轴1轴号,隔膜放卷纠偏 
	SlaveNo2:=AxiseNo.AxisName.SEPTAdeviation2 , //从轴2轴号，隔膜低部纠偏
	MasterValue:=100 ,//主轴速度 
	RecDevagree:=TRUE , //纠偏允许
	RecDevEqupos:=Mach_Control.DT_b.RecDevEqupos , //纠偏传感器平衡位置
	RecDevValueSet:=Par.stDT_date.RecDevValueSet , //纠偏偏差值设置
	RecDevPV:=Mach_Control.DT_b.RecDevPV , //纠偏传感器当前值
	RecDevSpeedCoe:=Par.stDT_date.RecDevSpeedCoe , //纠偏速度系数
	CWW:=Mach_Control.DT_b.CWW , //纠偏方向选择
	AxisPos_H:=Par.stDT_date.fRectifyMaxValue , //从轴纠偏行程上限
	AxisPos_L:=Par.stDT_date.fRectifyMinValue , //从轴纠偏行程下降
	RecDevSpeed=> , //从轴的速度
	Error=> );//错误报警
	
Rectifydev_V1.RecDevSpeed;



Mach_Control.DT_b.Error[9]:= Rectifydev_V1.Error[0];//纠偏凸轮耦合失败报警
Mach_Control.DT_b.Error[10]:=Rectifydev_V1.Error[1];//纠偏左限位报警
Mach_Control.DT_b.Error[11]:=Rectifydev_V1.Error[2];//纠偏右限位报警

*)
END_ACTION

ACTION _04Tension_Auto:

(******************************************************隔膜张力V2**SJ*****************************************************************************************)
Mach_Control.DT_b.fWindDiameter ;//放卷轴当前卷径
//par.stDT_date.Width:=102.7;
fbTensionGM(
		bReset:=                       stSysState.bReset   , 
		bCcw:=                         fbTensionGM.bCcw , //放卷方向选择
		fDanserDegree:=          Mach_Control.DT_b.TenAnglePos, //摆杆当前角度
		PidSwitch:=                   Mach_Control.DT_b.PidSwitch , //被动放卷选择   默认为TRUE，当为FALSE时摆杆偏离平衡位置时，不进行被动放卷
		bTenExecute:=              Mach_Control.DT_b.bTenExecute , //张力启动  AND arrCyCtrl[arrCyNo.CylinderName.PoleInflationCy].Io.DOStatus1
	    bStudyExecute:=           Mach_Control.DT_b.bStudyExecute , //张力学习
		
		fYDLength:=                 par.stDT_date.Width , //压力外边宽
		Ca_Quantited:=             Mach_Control.Ca_b.Ca_Quantited , 
		An_Quantited:=             Mach_Control.An_b.An_Quantited ,    
		fDancerMinPos:=           par.stDT_date.fDancerMinPos , //摆杆最小角度
		fDancerMaxPos:=          par.stDT_date.fDancerMaxPos ,  //摆杆最大角度
		fDanceBlancePos:=         par.stDT_date.fDanceBlancePos , //摆杆平衡位置
		FJ_Gemo:= 0.01, 
		fDiaMax:=220 , 
		fDiaMin:=80 , 
	    iGMMoveCount:=          Mach_Control.DT_b.TeniGMMoveCount ,//隔膜同步拉伸次数 
		
		bReady=>                        Mach_Control.DT_b.bTenReady , //张力准备好
		bTensionOK=>                 Mach_Control.DT_b.bTensionOK  , //张力OK 
		fWindDiameterTemp=>      Mach_Control.DT_b.fWindDiameter,//实时卷径
		bError=>                         Mach_Control.DT_b.Error[45],//张力报警 ???????????????
	
		Master:=                          arrAxis[AxiseNo.VirAxisName.VirDriver] , //放卷虚轴
		SlaveU:=                           arrAxis[AxiseNo.AxisName.SEPTAunwinding] , //放卷轴
		TimerAxis:=                       arrAxis[AxiseNo.VirAxisName.VirTimeWind],  //时间轴 
		Table:=                            Par.stDT_date.TensionTable , 
		Cache:=                              AxiseNo.AxisName.SEPTATCache );
	

IF NOT Mach_Control.DT_b.bTenReady AND NOT Mach_Control.DT_b.bTensionOK AND NOT Mach_Control.DT_b.bTenExecute THEN
	Mach_Control.DT_b.Error_tips[5]:=TRUE;////张力未准备好
ELSIF  Mach_Control.DT_b.bTenReady THEN
	Mach_Control.DT_b.Error_tips[5]:=FALSE ;////张力未准备好
END_IF		
		
//隔膜同步拉膜计数
rtGMMoveCount(CLK:= Mach_Control.DT_b.bTensionOK AND  NOT An_OverNGMark AND NOT Ca_OverNGMark AND
                                   arrAxis[AxiseNo.AxisName.SEPTATCache].Status.Coupled  AND
								   arrAxis[AxiseNo.AxisName.SEPTATLine].Status.Coupled AND 
                                   arrAxis[AxiseNo.VirAxisName.VirMain].Status.Moving  AND
								 (arrAxis[AxiseNo.VirAxisName.VirMain].NcToPlc.ModuloSetPos>=354 AND arrAxis[AxiseNo.VirAxisName.VirMain].NcToPlc.ModuloSetPos<=359));
IF rtGMMoveCount.Q THEN
    Mach_Control.DT_b.TeniGMMoveCount:=Mach_Control.DT_b.TeniGMMoveCount+1;
	fbTensionGM.fUsedLen:=fbTensionGM.fUsedLen+par.stDT_date.Width;
		//IF NOT Blueflaging THEN
		//		Par.stDT_date.HMI_Count[1]:=Par.stDT_date.HMI_Count[1]+0.1026;//拉膜长度
		//END_IF
END_IF

(*
IF 6016<=DP_Step0 AND DP_Step0<6050 THEN
	iTargetTorqueTest:=REAL_TO_INT(Par.stDT_date.iTargetTorqueHMI*LIMIT(0.3,Par.stDT_date.HMI_CountSet[2],1)); 
ELSE
	iTargetTorqueTest:=Par.stDT_date.iTargetTorqueHMI;
END_IF
*)

rtFlgGMEndIng(CLK:=bFlgGMEndIng , Q=> );//拉膜中
ftFlgGMEndIng(CLK:=bFlgGMEndIng , Q=> );//拉膜中

IF  rtFlgGMEndIng.Q  THEN
	fGMEndSatrtPos:=arrAxis[AxiseNo.AxisName.TailCurlLine].NcToPlc.ActPos;
END_IF

IF  ftFlgGMEndIng.Q  THEN
	fGMEndLength:=arrAxis[AxiseNo.AxisName.TailCurlLine].NcToPlc.ActPos-fGMEndSatrtPos;
END_IF


Mach_Control.Ca_b.Ca_Quantited;

//一键启动张力
rTension_Start(CLK:=Mach_Control.DT_b	.rTension_Start , Q=> );


//检测隔膜换卷
rtGMBtn(CLK:=arrCyCtrl[arrCyNo.CylinderName.PoleInflationCy].Io.DOStatus1 , Q=> );//涨紧
rtGMBtn2(CLK:=arrCyCtrl[arrCyNo.CylinderName.PoleInflationCy].Io.DOStatus2 , Q=> );//松开

IF rtGMBtn.Q THEN  
  
	iGMCheckSetp:=10;
END_IF

IF rtGMBtn2.Q THEN    
   	bFlgGMPulling:=FALSE;
	Mach_Control.DT_b.DT_QLqr:=FALSE;
   	iWindDiameterRecord2:=Mach_Control.DT_b.fWindDiameter;
	iGMCheckSetp:=0;
END_IF



CASE iGMCheckSetp OF
	
10:
   iWindDiameterRecord1:=Mach_Control.DT_b.fWindDiameter;
   //fGMLengthRecord:=ABS( FC_AngleToLength(arrAxisCtrl[AxiseNo.AxisName.SEPTAunwinding].Status.fActPos,sFB_TensionGMV2_1.fWindDiameterTemp) ) ;
   iGMCheckSetp:=20; 
20:
   IF ABS(iWindDiameterRecord1-iWindDiameterRecord2) >=50 AND   Mach_Control.U.DT_iMode=3   THEN
      iGMCheckSetp:=100;
   ELSE
	  iGMCheckSetp:=666;
   END_IF
 100: 
    bFlgGMPulling:=TRUE;
	Mach_Control.DT_b.DT_QLqr:=TRUE;
    iGMCheckSetp:=110; 
110:
	IF Mach_Control.DT_b.ClearCount THEN   // OR (Mach_Control.An_b.An_Quantited=0 AND Mach_Control.Ca_b.Ca_Quantited=0 )
		    	bFlgGMPulling:=FALSE;
			Mach_Control.DT_b.DT_QLqr:=FALSE;
			iGMCheckSetp:=667;	
	END_IF
END_CASE



rDtUse[2](CLK:=Mach_Control.U.DT_iMode=1 );//AND NOT  Mach_Control.DT_b.bTensionOK 
IF rDtUse[2].Q THEN
	iTensionAutoStep:=10;
END_IF
fDtUse[2](CLK:=Mach_Control.U.DT_iMode=1 );//叠台下降沿
IF fDtUse[2].Q THEN
	iTensionAutoStep:=0;
END_IF
//自动启动时叠台自动上张力
CASE iTensionAutoStep OF//叠台自动启动时张力自动步
10:
	IF Mach_Control.DT_b.bTensionOK THEN
		iTensionAutoStep:=6666;
	ELSE
		iTensionAutoStep:=50;
	END_IF
50:
	IF NOT arrCyCtrl[arrCyNo.CylinderName.PoleInflationCy].Io.DOStatus1 THEN
		 arrCyCtrl[arrCyNo.CylinderName.PoleInflationCy].Io.DOStatus1:=TRUE;
	ELSE
		iTensionAutoStep:=100;
	END_IF
100:
	tDtUse[1](IN:=arrCyCtrl[arrCyNo.CylinderName.PoleInflationCy].Io.DOStatus1 , PT:=T#0.5S , Q=> , ET=> );
	IF NOT arrCyCtrl[arrCyNo.CylinderName.PoleInflationCy].Io.DOStatus1 THEN
		arrCyCtrl[arrCyNo.CylinderName.PoleInflationCy].Cmd.bON:=TRUE;
		arrCyCtrl[arrCyNo.CylinderName.PoleInflationCy].Cmd.bOFF:=FALSE;
	END_IF
	IF tDtUse[1].Q THEN
		iTensionAutoStep:=200;	
	END_IF
200://开张力
	IF Mach_Control.DT_b.bTenReady THEN
		Mach_Control.DT_b.bTenExecute:=TRUE;
		iTensionAutoStep:=300;
	ELSE
		Mach_Control.DT_b.Error_tips[5]:=TRUE;////张力未准备好
	END_IF	
300:
	IF Mach_Control.DT_b.bTensionOK THEN   //张力OK 
		iTensionAutoStep:=6666;	
	END_IF
END_CASE




//卷径转换长度，单位米
 fDiameterORLength(	D1:=Mach_Control.DT_b.fWindDiameter ,
					R1:=Par.stDT_date.fInsideDiameter , 
					T1:=Par.stDT_date.SEPTA_Thickness ,
					OUT1=>Mach_Control.DT_b.fWindLength_M );



//Par.stDT_date.iTargetTorqueHMI:=REAL_TO_INT((par.stDT_date.fTenset-par.stDT_date.fTen_B)/par.stDT_date.fTen_K);


(*

//隔膜张力
sFB_TensionGMV2_1(
	bReset:=stSysState.bReset  , //复位
	bCcw:=sFB_TensionGMV2_1.bCcw , //放卷方向选择
	fDanserDegree:= Mach_Control.DT_b.TenAnglePos, //摆杆当前角度
	fWindDiameter:=Mach_Control.DT_b.fWindDiameter , //放卷轴当前卷径
	PidSwitch:=Mach_Control.DT_b.PidSwitch , //被动放卷选择   默认为TRUE，当为FALSE时摆杆偏离平衡位置时，不进行被动放卷
	bTenExecute:=Mach_Control.DT_b.bTenExecute AND arrCyCtrl[arrCyNo.CylinderName.PoleInflationCy].Status.ONState, //张力启动
	bStudyExecute:=Mach_Control.DT_b.bStudyExecute , //张力学习
	fStudyDiameter:=par.stDT_date.fStudyDiameter  , //学习时隔膜的卷径
	fYDLength:=par.stDT_date.Width , //压力外边宽
	Ca_Quantited:=Mach_Control.Ca_b.Ca_Quantited , //压力外边宽
	fDancerMinPos:=par.stDT_date.fDancerMinPos , //摆杆最小角度
	fDancerMaxPos:=par.stDT_date.fDancerMaxPos ,  //摆杆最大角度
	fDanceBlancePos:=par.stDT_date.fDanceBlancePos , //摆杆平衡位置
	bReady=>Mach_Control.DT_b.bTenReady , //张力准备好
	bTensionOK=>Mach_Control.DT_b.bTensionOK  , //张力OK
	bError=> , 
	iGMMoveCount:=Mach_Control.DT_b.TeniGMMoveCount ,//隔膜同步拉伸次数
	fGMEndLength:=fGMEndLength,
	Master:=arrAxis[AxiseNo.VirAxisName.VirDriver] , //放卷虚轴
	Slave:=arrAxis[AxiseNo.AxisName.SEPTAunwinding] , //放卷轴
	TimerAxis:= arrAxis[AxiseNo.VirAxisName.VirTimeWind],  //时间轴
	Table:=Par.stDT_date.TensionTable  );	
	
     sFB_TensionGMV2_1.fDiameterCalculate;
	  sFB_TensionGMV2_1.fWindDiameterTemp;
	
	//隔膜同步拉膜计数
rtGMMoveCount(CLK:=        Mach_Control.DT_b.bTensionOK     AND 
      arrAxis[AxiseNo.AxisName.SEPTATCache] .Status.Coupled    AND 
          arrAxis[AxiseNo.AxisName.SEPTATLine].Status.Coupled    AND 
             arrAxis[AxiseNo.VirAxisName.VirMain].Status.Moving   AND   ( arrAxis[AxiseNo.VirAxisName.VirMain].NcToPlc.ModuloSetPos>=354 AND   arrAxis[AxiseNo.VirAxisName.VirMain].NcToPlc.ModuloSetPos<=359  )
 , Q=> );
IF rtGMMoveCount.Q THEN
    Mach_Control.DT_b.TeniGMMoveCount:=Mach_Control.DT_b.TeniGMMoveCount+1;
END_IF


rtFlgGMEndIng(CLK:=bFlgGMEndIng , Q=> );//拉膜中
ftFlgGMEndIng(CLK:=bFlgGMEndIng , Q=> );//拉膜中

IF  rtFlgGMEndIng.Q  THEN
	fGMEndSatrtPos:=arrAxis[AxiseNo.AxisName.TailCurlLine].NcToPlc.ActPos;
END_IF

IF  ftFlgGMEndIng.Q  THEN
	fGMEndLength:=arrAxis[AxiseNo.AxisName.TailCurlLine].NcToPlc.ActPos-fGMEndSatrtPos;
END_IF


Mach_Control.Ca_b.Ca_Quantited;

//一键启动张力
rTension_Start(CLK:=Mach_Control.DT_b	.rTension_Start , Q=> );


//检测隔膜换卷
rtGMBtn(CLK:=arrCyCtrl[arrCyNo.CylinderName.PoleInflationCy].Io.DOStatus1 , Q=> );//涨紧
rtGMBtn2(CLK:=arrCyCtrl[arrCyNo.CylinderName.PoleInflationCy].Io.DOStatus2 , Q=> );//松开

IF rtGMBtn.Q THEN  
  
	iGMCheckSetp:=10;
END_IF

IF rtGMBtn2.Q THEN    
   	bFlgGMPulling:=FALSE;
	Mach_Control.DT_b.DT_QLqr:=FALSE;
   	iWindDiameterRecord2:=Mach_Control.DT_b.fWindDiameter;
	iGMCheckSetp:=0;
END_IF



CASE iGMCheckSetp OF
	
10:
   iWindDiameterRecord1:=Mach_Control.DT_b.fWindDiameter;
   //fGMLengthRecord:=ABS( FC_AngleToLength(arrAxisCtrl[AxiseNo.AxisName.SEPTAunwinding].Status.fActPos,sFB_TensionGMV2_1.fWindDiameterTemp) ) ;
   iGMCheckSetp:=20; 
20:
   IF ABS(iWindDiameterRecord1-iWindDiameterRecord2) >=50 AND   Mach_Control.U.DT_iMode=3   THEN
      iGMCheckSetp:=100;
   ELSE
	  iGMCheckSetp:=666;
   END_IF
 100: 
    bFlgGMPulling:=TRUE;
	Mach_Control.DT_b.DT_QLqr:=TRUE;
    iGMCheckSetp:=110; 
110:
	IF Mach_Control.DT_b.ClearCount THEN   // OR (Mach_Control.An_b.An_Quantited=0 AND Mach_Control.Ca_b.Ca_Quantited=0 )
		    bFlgGMPulling:=FALSE;
			Mach_Control.DT_b.DT_QLqr:=FALSE;
			iGMCheckSetp:=667;	
	END_IF
END_CASE


(*
CASE iGMCheckSetp OF
	
10:
   iCa_QuantitedRecord:=Mach_Control.Ca_b.Ca_Quantited;
   fGMLengthRecord:=ABS( FC_AngleToLength(arrAxisCtrl[AxiseNo.AxisName.SEPTAunwinding].Status.fActPos,sFB_TensionGMV2_1.fWindDiameterTemp) ) ;
   iGMCheckSetp:=20; 
20:
  IF  Mach_Control.DT_b.bTensionOK  AND 
	  iCa_QuantitedRecord=Mach_Control.Ca_b.Ca_Quantited AND   
      ABS( FC_AngleToLength(arrAxisCtrl[AxiseNo.AxisName.SEPTAunwinding].Status.fActPos,sFB_TensionGMV2_1.fWindDiameterTemp) ) - fGMLengthRecord >=500 AND 
	  Mach_Control.U.DT_iMode=3  THEN    //处于拉膜中
        iGMCheckSetp:=100; 
  END_IF

  IF  Mach_Control.DT_b.bTensionOK  AND 
	  iCa_QuantitedRecord<>Mach_Control.Ca_b.Ca_Quantited  THEN  //只是气涨轴动作无换卷
        iGMCheckSetp:=666; 
  END_IF
  
 
 100: 
    bFlgGMPulling:=TRUE;
    iGMCheckSetp:=667; 
 
 
 

END_CASE

*)






*)
END_ACTION

ACTION All_GoHome:
	f_AllGohome(CLK:=AllGohome_Hbtn ,Q=> );
	r_AllGohome(CLK:=AllGohome_Hbtn ,Q=> );	
	IF r_AllGohome.Q THEN
	AllGohomeTon[1].IN:=FALSE;
	AllGohomeTon[2].IN:=FALSE;
	AllGohomeTon[3].IN:=FALSE;
	TJIniti_Done:=FALSE;
	WZIniti_Done:=FALSE;
	Mach_Control.DT_b.DTIniti_Done:=FALSE;
	An_GohomeDone:=FALSE;
	Ca_GohomeDone:=FALSE;
	Ca_BeltGohomeDone:=FALSE;
	Step_InitCaDT0:=0;
	Step_InitAnDT:=0;
	Step_InitDT:=0;
	Step_InitCaDT:=0;
	TailCurlStep1:=0;
	StickerStep0:=0;
	AllGohomeStep:=10;
	Mach_Control.DT_b.ClearCount:=TRUE;
	END_IF	
	AllGohomeTon[1](PT:=T#10S);
	AllGohomeTon[2](PT:=T#10S);
	AllGohomeTon[3](PT:=T#5S);
	
IF Mach_Control.Ca_b.Error[19]//负极回原点超时报警
OR Mach_Control.Ca_b.Error[20]//负极皮带回原点超时报警
OR Mach_Control.An_b.Error[19]//负极回原点超时报警
OR Mach_Control. DT_b.Error[23]//叠台回原点超时报警
OR Mach_Control.WJ_b.Error[19]//尾卷回原点超时报警
OR Mach_Control.TJ_b.Error[8]  //贴胶回原超时报警
OR Step_InitCaDT0=9999 
OR Step_InitAnDT=9999 
OR Step_InitDT=9999
OR Step_InitCaDT=9999
OR TailCurlStep1=9999
OR StickerStep0=9999
THEN
	AllGohomeStep:=999;
END_IF
AllGohome_Done:=Mach_Control.WJ_b.WZIniti_Done AND Mach_Control.DT_b.DT_init_OK AND Mach_Control.Ca_b.Ca_BeltGohomeDone AND Mach_Control.TJ_b.TJIniti_Done;
CASE AllGohomeStep OF
10:
	IF f_AllGohome.Q THEN
	Mach_Control.DT_b.ClearCount:=FALSE;
	Mach_Control.WJ_b.WZIniti_Hbtn:=TRUE;
	AllGohomeStep:=20;
	END_IF
	
20:
	Mach_Control.WJ_b.WZIniti_Hbtn:=FALSE;
	AllGohomeStep:=30;

30:
	AllGohomeTon[1].IN:=TRUE;
	IF AllGohomeTon[1].Q AND Mach_Control.WJ_b.WZIniti_Done THEN
	Mach_Control.DT_b.ALLIniti_Hbtn:=TRUE;
	AllGohomeStep:=40;	
	END_IF
	
40:
	AllGohomeTon[1].IN:=FALSE;
	Mach_Control.DT_b.ALLIniti_Hbtn:=FALSE;
	AllGohomeStep:=50;	

50:
	AllGohomeTon[2].IN:=TRUE;
	IF AllGohomeTon[2].Q AND Mach_Control.DT_b.DT_init_OK THEN
	Mach_Control.Ca_b.Ca_BeltGohomeHMI:=TRUE;
	Mach_Control.TJ_b.TJIniti_Hbtn:=TRUE;
	AllGohomeStep:=60;	
	END_IF
	
60:
	AllGohomeTon[2].IN:=FALSE;
	Mach_Control.Ca_b.Ca_BeltGohomeHMI:=FALSE;
	Mach_Control.TJ_b.TJIniti_Hbtn:=FALSE;
	AllGohomeStep:=70;

70:
	AllGohomeTon[3].IN:=TRUE;
	IF AllGohomeTon[3].Q AND Mach_Control.Ca_b.Ca_BeltGohomeDone AND Mach_Control.TJ_b.TJIniti_Done THEN
	AllGohomeStep:=80;	
	END_IF	
80:
AllGohomeTon[3].IN:=FALSE;
AllGohomeStep:=888;	
END_CASE
END_ACTION

ACTION An_Alarm:


//报警时间
An_AlarmTon[1](IN:= , PT:=T#80MS , Q=> , ET=> );//正极送片搬运升降有真空信号，无极片报警延时
An_AlarmTon[2](IN:= , PT:=T#80MS , Q=> , ET=> );//正极送片搬运升降有极片，无真空信号报警延时
An_AlarmTon[3](IN:= , PT:=T#150MS , Q=> , ET=> );//正极叠台搬运升降有真空信号，无极片报警延时
An_AlarmTon[4](IN:= , PT:=T#80MS , Q=> , ET=> );//正极叠台搬运升降有极片，无真空信号报警延时
An_AlarmTon[5](IN:= , PT:=T#80MS , Q=> , ET=> );//正极纠偏平台有真空信号，无极片报警延时
An_AlarmTon[6](IN:= , PT:=T#150MS , Q=> , ET=> );//正极纠偏平台有极片，无真空信号报警延时
An_AlarmTon[7](IN:= , PT:=T#80MS , Q=> , ET=> );//正极纠偏平台连续NG
An_AlarmTon[8](IN:= , PT:=T#80MS , Q=> , ET=> );
An_AlarmTon[9](IN:= , PT:=T#300MS , Q=> , ET=> );
An_AlarmTon[10](IN:= , PT:=T#400MS , Q=> , ET=> );//
An_AlarmTon[11](IN:= , PT:=T#300MS , Q=> , ET=> );//正极极片对齐度检测返回结果超时
An_AlarmTon[12](IN:= , PT:=T#400MS , Q=> , ET=> );//正极CCD纠偏平台检测返回结果超时
An_AlarmTon[13](IN:=AnCCDMark , PT:=T#50MS , Q=> , ET=> );//正极CCD纠偏平台检测返回结果超时

An_AlarmTon[15](IN:= , PT:=T#50MS , Q=> , ET=> );//正极CCD纠偏平台检测返回结果超时
An_AlarmTon[16](IN:= , PT:=T#50MS , Q=> , ET=> );//正极CCD纠偏平台检测返回结果超时
An_AlarmTon[17](IN:=NOT Mach_Control.se.AnNGboxsensor , PT:=T#5S , Q=> , ET=> );//正极NG料盒料满

rAnUse[2](CLK:=Mach_Control.An_b.An_CCDStart AND NOT   Mach_Control.An_b.Demarcateing , Q=> );
rAnUse[3](CLK:=Par.stDT_date.An_Rectifydev_Btn , Q=> );
rAnUse[4](CLK:=arrCyCtrl[arrCyNo.ElectValveName.AnCarryingVacuum].Io.DOStatus1 , Q=> );  
rAnUse[5](CLK:= NOT arrCyCtrl[arrCyNo.ElectValveName.AnDTCarryingVacuum].Io.DOStatus1 , Q=> );

//Mach_Control.An_b.Error[1] :=TRUE;//正极送片搬运升降有真空信号，无极片报警
//Mach_Control.An_b.Error[2] :=TRUE;//正极送片搬运升降有极片，无真空信号报警
//Mach_Control.An_b.Error[3]:=TRUE;//正极叠台搬运升降在叠片过程中真空报警，请检查叠台是否掉片
//Mach_Control.An_b.Error[4] :=TRUE;//正极叠台搬运升降有极片，无真空信号报警
//Mach_Control.An_b.Error[5]:=TRUE;//正极纠偏平台有真空信号，无极片报警
//Mach_Control.An_b.Error[6]:=TRUE;//正极纠偏平台有极片，无真空信号报警
//Mach_Control.An_b.Error[7]:=TRUE;//纠偏CCD拍照完成IO信号未给出
//Mach_Control.An_b.Error[8]  ;//CCD标定NG
//Mach_Control.An_b.Error[9]  ;
//Mach_Control.An_b.Error[10]  ;
//Mach_Control.An_b.Error[11]:=TRUE;//正极有凸轮耦合报警
//Mach_Control.An_b.Error[12]:=TRUE;//正极NG收纳盒满料报警
//Mach_Control.An_b.Error[13];
//Mach_Control.An_b.Error[14]:=TRUE;//正极防撞感应信号报警
//Mach_Control.An_b.Error[15]
//Mach_Control.An_b.Error[16]
//Mach_Control.An_b.Error[17]
//Mach_Control.An_b.Error[18] :=TRUE;//正极CCD纠偏平台检测返回结果超时
// Mach_Control.An_b.Error[19]:=TRUE;//正极回原点超时报警
// Mach_Control.An_b.Error[20];
//Mach_Control.An_b.Error[21]:=TRUE;//正极纠偏平台连续NG
//Mach_Control.An_b.Error[22]:=TRUE;//正极叠台搬运升降真空报警，电芯上有片，请拿掉
//Mach_Control.An_b.Error[23]:=TRUE;//正极叠台搬运升降真空报警，电芯上无掉片
//Mach_Control.An_b.Error[24] ////正极纠偏平台NG片未排掉报警，请拿掉
//Mach_Control.An_b.Error[25] ////正极极片对齐度检测返回结果超时
//Mach_Control.An_b.Error[26] ////正极搬运防撞软限位报警
//Mach_Control.An_b.Error[27]//    //正极极片对齐度检测返回结果无片报警
//Mach_Control.An_b.Error[28]//正极叠片完空叠隔膜时，正极叠片搬运机械手真空有信号、标记有极片报警,请拿掉极片
//Mach_Control.An_b.Error[29]:=TRUE;		//正极初始化时正极叠片搬运升降吸盘有真空报警
//Mach_Control.An_b.Error[30]:=TRUE;		//正极初始化时正极送片搬运升降吸盘有真空报警	

//Mach_Control.An_b.Error[32]:=TRUE;//正极送片搬运在叠片过程中真空报警
//Mach_Control.An_b.Error[33]:=FALSE;//纠偏平台有片，请拿走
//Mach_Control.An_b.Error[34]:=FALSE;//正极叠台搬运平移取片时真空报警,请确认纠偏台是否掉片
//Mach_Control.An_b.Error[35]:=TRUE;//正极纠偏台NG料盒料满报警
//Mach_Control.An_b.Error[36]:=TRUE;//正极纠偏纠偏CCD返回结果超时
//Mach_Control.An_b.Error[37]:=TRUE;//正极叠台搬运升降有真空信号，无极片报警
//Mach_Control.An_b.Error[38] :=TRUE;//正极叠台搬运升降有极耳无真空报警
//Mach_Control.An_b.Error[39] :=TRUE;//正极叠台搬运升降有极耳无真空报警
//Mach_Control.An_b.Error[40] S=AnOverNGcount>=3;//正极单张踢废连续NG
//Mach_Control.An_b.Error[41] :=TRUE;//正极机械手初始化时，叠台搬运升降不在避让位
Mach_Control.An_b.Error[40] S=AnOverNGcount>=3;//正极单张踢废连续NG

//NG料盒料满报警
	IF (*Par.stDT_date.An_Rectifydev_JS>=Par.stDT_date.An_Rectifydev_NGSet OR*) An_AlarmTon[17].Q THEN
		Mach_Control.An_b.Error[35]:=TRUE;//负极纠偏台NG料盒料满报警
	ELSE
		Mach_Control.An_b.Error[35]:=FALSE;//负极纠偏台NG料盒料满报警
	END_IF
	IF rAnUse[3].Q THEN
		Par.stDT_date.An_Rectifydev_JS:=0;
	END_IF



//正极初始化时有真空报警	
	IF Mach_Control.An_b.An_GohomeHMI THEN
		IF arrCyCtrl[arrCyNo.ElectValveName.AnDTCarryingVacuum].Status.ONState  THEN    
			Mach_Control.An_b.Error[29]:=TRUE;		//正极初始化时正极叠片搬运升降吸盘有真空报警
		END_IF
		IF arrCyCtrl[arrCyNo.ElectValveName.	AnCarryingVacuum	].Status.ONState THEN	
			Mach_Control.An_b.Error[30]:=TRUE;		//正极初始化时正极送片搬运升降吸盘有真空报警	
		END_IF		 
	END_IF	
(*
//正极送片搬运升降真空信号与有无极片标记不一致报警
An_AlarmTon[1].IN:=arrCyCtrl[arrCyNo.ElectValveName.AnCarryingVacuum].Io.DIOnSwitch AND NOT Mach_Control.An_b.An_CarryingFalg 
	AND NOT Mach_Control.U.EmptyRunMode AND NOT Mach_Control.An_b.Error[2]  AND NOT Blueflaging AND Mach_Control.U.DT_iMode=1;
		IF  An_AlarmTon[1].Q THEN
				Mach_Control.An_b.Error[1] :=TRUE;//正极送片搬运升降有真空信号，无极片报警
		END_IF
*)
//正极送片搬运升降有极片，无真空信号报警------取片过程中真空报警判断
An_AlarmTon[2].IN:=NOT arrCyCtrl[arrCyNo.ElectValveName.AnCarryingVacuum].Io.DIOnSwitch AND  Mach_Control.An_b.An_CarryingFalg  AND
	 arrAxisCtrl[AxiseNo.AxisName.AnCarryingUpDown].Status.fActPos<=(arrAxisPar[AxiseNo.AxisName.AnCarryingUpDown].arrTargetPoint[2]-5) 
	AND arrAxisCtrl[AxiseNo.AxisName.AnCarryingLine].Status.NoMoving AND NOT Mach_Control.U.EmptyRunMode ;
	IF  An_AlarmTon[2].Q THEN
			Mach_Control.An_b.Error[2] :=TRUE;//正极送片搬运升降有极片，无真空信号报警
			(*
			Mach_Control.An_b.An_CarryingFalg:=FALSE;
			arrCyCtrl[arrCyNo.ElectValveName.AnCarryingVacuum].Cmd.bOFF:=TRUE;//正极搬运升降取料真空关
			arrCyCtrl[arrCyNo.ElectValveName.AnCarryingVacuum].Cmd.bON:=FALSE;//正极搬运升降取料真空关
			arrCyCtrl[arrCyNo.ElectValveName.AnCarryingVacuumBark].Cmd.bON:=TRUE;//正极搬运升降取料破真空开
			arrCyCtrl[arrCyNo.ElectValveName.AnCarryingVacuumBark].Cmd.bOFF:=FALSE;//正极搬运升降取料破真空开
			*)
	END_IF
IF 	Mach_Control.An_b.Error[2]AND arrCyCtrl[arrCyNo.ElectValveName.AnCarryingVacuum].Io.DIOnSwitch AND  rAn_AlarmRest.Q  THEN
	Mach_Control.An_b.Error[2] :=FALSE;//正极送片搬运升降有极片，无真空信号报警
ELSIF Mach_Control.An_b.Error[2]AND NOT arrCyCtrl[arrCyNo.ElectValveName.AnCarryingVacuum].Io.DIOnSwitch AND  rAn_AlarmRest.Q  THEN
	arrCyCtrl[arrCyNo.ElectValveName.AnCarryingVacuum].Cmd.bOFF:=TRUE;//正极搬运升降取料真空关
	arrCyCtrl[arrCyNo.ElectValveName.AnCarryingVacuum].Cmd.bON:=FALSE;//正极搬运升降取料真空关
	arrCyCtrl[arrCyNo.ElectValveName.AnCarryingVacuumBark].Cmd.bON:=TRUE;//正极搬运升降取料破真空开
	arrCyCtrl[arrCyNo.ElectValveName.AnCarryingVacuumBark].Cmd.bOFF:=FALSE;//正极搬运升降取料破真空开
	An_StandbyStep1:=0;
	An_Step0:=0;
	An_Step1:=0;
	An_Step2:=0;
	An_Step3:=0;
	Mach_Control.An_b.Error[2] :=FALSE;//正极送片搬运升降有极片，无真空信号报警
	Mach_Control.An_b.An_CarryingFalg:=FALSE;
END_IF
	
	
	
	
	
//正极送片搬运在叠片过程中的真空信号判断
	An_AlarmTon[15].IN:=NOT arrCyCtrl[arrCyNo.ElectValveName.AnCarryingVacuum].Io.DIOnSwitch AND  Mach_Control.An_b.An_CarryingFalg 
	AND NOT Mach_Control.U.EmptyRunMode AND arrAxisCtrl[AxiseNo.AxisName.AnCarryingLine].Status.Moving	  
	 AND  arrAxisCtrl[AxiseNo.VirAxisName.VirMain].Status.fActPos<232 AND  arrAxisCtrl[AxiseNo.VirAxisName.VirMain].Status.fActPos>1   ;
	IF  An_AlarmTon[15].Q THEN
		CCD.AnRec.Finish.RectifyResult:=0;
		Mach_Control.An_b.Error[32] :=TRUE;//正极送片搬运升降有极片，无真空信号报警
		Mach_Control.An_b.An_CarryingFalg:=FALSE;
		arrCyCtrl[arrCyNo.ElectValveName.AnCarryingVacuum].Cmd.bOFF:=TRUE;//正极搬运升降取料真空关
		arrCyCtrl[arrCyNo.ElectValveName.AnCarryingVacuum].Cmd.bON:=FALSE;//正极搬运升降取料真空关
		arrCyCtrl[arrCyNo.ElectValveName.AnCarryingVacuumBark].Cmd.bON:=TRUE;//正极搬运升降取料破真空开
		arrCyCtrl[arrCyNo.ElectValveName.AnCarryingVacuumBark].Cmd.bOFF:=FALSE;//正极搬运升降取料破真空开
	END_IF
	IF Mach_Control.An_b.Error[32] AND rAn_AlarmRest.Q   THEN
		//CCD.AnRec.Finish.RectifyResult:=0;
		CCD.AnRec.Start.iPhotoDo:=1;//第二次拍照
		Mach_Control.An_b.An_CCDStart :=TRUE;//启动CCD拍照
	END_IF
	IF Mach_Control.An_b.Error[32] AND (CCD.AnRec.Finish.RectifyResult=3  OR  Mach_Control.U.CCD_ChosesHMI) AND rAn_AlarmRest.Q  THEN
		Mach_Control.An_b.Error[32]:=FALSE;
		Mach_Control.An_b.Error[33]:=FALSE;//纠偏平台有片，请拿走
	END_IF
	IF Mach_Control.An_b.Error[32] AND (CCD.AnRec.Finish.RectifyResult<>3  AND NOT   Mach_Control.U.CCD_ChosesHMI)THEN
		Mach_Control.An_b.Error[33]:=TRUE;//纠偏平台有片，请拿走
	END_IF
	
	
	
	
	
//正极叠片搬运升降真空信号与有无极片标记不一致报警
An_AlarmTon[3].IN:=(arrCyCtrl[arrCyNo.ElectValveName.AnDTCarryingVacuum].Io.DIOnSwitch OR Mach_Control.se.AnDTCarryingJROnSwitch)
    AND NOT Mach_Control.An_b.An_DPCarryingFalg AND Mach_Control.U.DT_iMode=1 
	AND NOT Mach_Control.U.EmptyRunMode AND (An_Step2=0 OR An_Step2=6666) AND NOT Mach_Control.An_b.Error[4] AND iEmptyFoldStep[1]=0 
	AND arrAxisCtrl[AxiseNo.AxisName.AnDTCarryingUpDown].Status.fActPos<=(arrAxisPar[AxiseNo.AxisName.AnDTCarryingUpDown].arrTargetPoint[2]-5)  
	AND DP_Step0<1000 AND DP_Step0>3100;
	IF  An_AlarmTon[3].Q THEN
		IF arrCyCtrl[arrCyNo.ElectValveName.AnDTCarryingVacuum].Io.DIOnSwitch THEN
			Mach_Control.An_b.Error[3]:=TRUE;//正极叠台搬运升降有真空信号，无极片报警
		END_IF
        IF 	Mach_Control.se.AnDTCarryingJROnSwitch THEN
			Mach_Control.An_b.Error[37]:=TRUE;//正极叠台搬运升降有真空信号，无极片报警
		END_IF
	END_IF

	
//正极叠台搬运升降有极片，无真空信号报警-------叠片搬运平移取片过程真空检测
An_AlarmTon[16].IN:=(NOT arrCyCtrl[arrCyNo.ElectValveName.AnDTCarryingVacuum].Io.DIOnSwitch OR NOT Mach_Control.se.AnDTCarryingJROnSwitch)
     AND  Mach_Control.An_b.An_DPCarryingFalg  AND (An_Step2=0 OR An_Step2=6666) AND
	arrAxisCtrl[AxiseNo.AxisName.AnDTCarryingUpDown].Status.fActPos<=(arrAxisPar[AxiseNo.AxisName.AnDTCarryingUpDown].arrTargetPoint[2]-5)  
	AND  arrAxisCtrl[AxiseNo.AxisName.AnDTCarryingLine].Status.NoMoving AND NOT Mach_Control.U.EmptyRunMode AND iEmptyFoldStep[1]=0 
	AND (DP_Step0<1000 OR DP_Step0>3100)  ;//
	IF  An_AlarmTon[16].Q THEN
		//CCD.AnRec.Finish.RectifyResult:=0;//拍照结果清零
		IF NOT arrCyCtrl[arrCyNo.ElectValveName.AnDTCarryingVacuum].Io.DIOnSwitch THEN
		   Mach_Control.An_b.Error[34] :=TRUE;//正极叠台搬运升降有极片，无真空信号报警
		END_IF  
		IF NOT Mach_Control.se.AnDTCarryingJROnSwitch THEN
           Mach_Control.An_b.Error[39] :=TRUE;//正极叠台搬运升降有极耳无真空报警
        END_IF   
		Mach_Control.An_b.An_DPCarryingFalg:=FALSE;
		arrCyCtrl[arrCyNo.ElectValveName.AnDTCarryingVacuum].Cmd.bOFF:=FALSE;//正极叠片搬运升降真空关
		arrCyCtrl[arrCyNo.ElectValveName.AnDTCarryingVacuum].Cmd.bON:=TRUE;//正极叠片搬运升降真空关
		//arrCyCtrl[arrCyNo.ElectValveName.AnDTCarryingVacuumBark].Cmd.bON:=TRUE;//正极叠片搬运破真空开
		//arrCyCtrl[arrCyNo.ElectValveName.AnDTCarryingVacuumBark].Cmd.bOFF:=FALSE;//正极叠片搬运破真空关
	END_IF
//叠台搬运平移在取片过程中报警时，纠偏平台拍照有无片来确定是否掉片到纠偏平台
	IF (Mach_Control.An_b.Error[34] OR Mach_Control.An_b.Error[39]) AND rAn_AlarmRest.Q  THEN
		//CCD.AnRec.Finish.RectifyResult:=0;//拍照结果清零
		Mach_Control.An_b.An_CCDStart :=TRUE;//启动CCD拍照
		CCD.AnRec.Start.iPhotoDo:=1;//启动CCD第二次拍照
	END_IF
	IF (Mach_Control.An_b.Error[34] OR Mach_Control.An_b.Error[39]) AND (CCD.AnRec.Finish.RectifyResult=3  OR  Mach_Control.U.CCD_ChosesHMI) AND rAn_AlarmRest.Q  THEN
		Mach_Control.An_b.Error[34]:=FALSE;//叠台升降取片过程中真空报警，
		Mach_Control.An_b.Error[39]:=FALSE;//叠台升降取片过程中真空报警，
		Mach_Control.An_b.Error[33]:=FALSE;//纠偏平台有片，请拿走
	ELSIF( Mach_Control.An_b.Error[34] OR Mach_Control.An_b.Error[39]) AND (CCD.AnRec.Finish.RectifyResult<>3  AND NOT   Mach_Control.U.CCD_ChosesHMI)THEN
		Mach_Control.An_b.Error[33]:=TRUE;//纠偏平台有片，请拿走
	END_IF
	






	
	
//正极叠台搬运升降有极片，无真空信号报警-------叠片搬运平移叠片过程真空检测
An_AlarmTon[4].IN:=(NOT arrCyCtrl[arrCyNo.ElectValveName.AnDTCarryingVacuum].Io.DIOnSwitch OR NOT Mach_Control.se.AnDTCarryingJROnSwitch)
     AND  Mach_Control.An_b.An_DPCarryingFalg  AND (An_Step2=0 OR An_Step2=6666) AND
	 arrAxisCtrl[AxiseNo.VirAxisName.VirMain].Status.fActPos<232 AND  arrAxisCtrl[AxiseNo.VirAxisName.VirMain].Status.fActPos>1  AND NOT Mach_Control.U.EmptyRunMode
	AND  arrAxisCtrl[AxiseNo.AxisName.AnDTCarryingLine].Status.Moving	 ;//
	IF  An_AlarmTon[4].Q THEN
		//Mach_Control.DT_b.OverhandResult:=0;
		IF NOT arrCyCtrl[arrCyNo.ElectValveName.AnDTCarryingVacuum].Io.DIOnSwitch THEN
		  Mach_Control.An_b.Error[4] :=TRUE;//正极叠台搬运升降有极片，无真空信号报警
	    END_IF
		IF  NOT Mach_Control.se.AnDTCarryingJROnSwitch THEN
		  Mach_Control.An_b.Error[38] :=TRUE;//正极叠台搬运升降有极耳无真空报警
		END_IF
		An_Number:=TRUE;
		Mach_Control.An_b.An_DPCarryingFalg:=FALSE;
		arrCyCtrl[arrCyNo.ElectValveName.AnDTCarryingVacuum].Cmd.bOFF:=FALSE;//正极叠片搬运升降真空关
		arrCyCtrl[arrCyNo.ElectValveName.AnDTCarryingVacuum].Cmd.bON:=TRUE;//正极叠片搬运升降真空关
		//arrCyCtrl[arrCyNo.ElectValveName.AnDTCarryingVacuumBark].Cmd.bON:=TRUE;//正极叠片搬运破真空开
		//arrCyCtrl[arrCyNo.ElectValveName.AnDTCarryingVacuumBark].Cmd.bOFF:=FALSE;//正极叠片搬运破真空关
	END_IF
	
	//正极叠台搬运升降真空报警，电芯上有片，请拿掉
	An_AlarmTon[8].IN:=(Mach_Control.An_b.Error[4] OR Mach_Control.An_b.Error[38]) AND Mach_Control.DT_b.OverhandResult<>3 AND NOT Mach_Control.U.CCD_ChosesHMI ;
	IF  An_AlarmTon[8].Q THEN
		Mach_Control.An_b.Error[22]:=TRUE;//正极叠台搬运升降真空报警，电芯上有片，请拿掉
	END_IF
	IF fAn_AlarmRest.Q AND  Mach_Control.An_b.Error[22] AND arrAxisCtrl[AxiseNo.VirAxisName.VirMain].Status.fActPos<1  THEN
		Mach_Control.DT_b.OverhandResult:=0;
		CCD.Over.Start.iPhotoDo:=2;
		Mach_Control.DT_b.CDD_OverStart:=TRUE;
	END_IF

	IF Mach_Control.An_b.Error[22] AND Mach_Control.DT_b.OverhandResult=3  AND rAn_AlarmRest.Q THEN
		Mach_Control.An_b.Error[22]:=FALSE;//复位电芯有片报警
		Mach_Control.DT_b.OverhandResult:=0;
	END_IF
	
	//正极叠台搬运升降真空报警，电芯上无掉片
	An_AlarmTon[9].IN:=(Mach_Control.An_b.Error[4] OR Mach_Control.An_b.Error[38] )AND Mach_Control.DT_b.OverhandResult=3 AND NOT Mach_Control.U.CCD_ChosesHMI ;
	IF  An_AlarmTon[9].Q THEN
		Mach_Control.An_b.Error[23]:=TRUE;//正极叠台搬运升降真空报警，电芯上无掉片
	END_IF

	
	

//正极纠偏平台真空信号与有无极片标记不一致报警
An_AlarmTon[5].IN:=arrCyCtrl[arrCyNo.ElectValveName.AndeviationVacuum].Io.DIOnSwitch AND NOT Mach_Control.An_b.An_deviationFalg 
	AND NOT Mach_Control.U.EmptyRunMode AND arrAxisCtrl[AxiseNo.AxisName.AnDTCarryingUpDown].Status.Homed 
	AND arrAxisCtrl[AxiseNo.AxisName.AnDTCarryingUpDown].Status.fActPos<=(arrAxisPar[AxiseNo.AxisName.AnDTCarryingUpDown].arrTargetPoint[4]+5) 
	AND iEmptyFoldStep[1]=0 AND (DP_Step0<1000 OR DP_Step0>3100) ;
	IF  An_AlarmTon[5].Q THEN
		Mach_Control.An_b.Error[5]:=TRUE;//正极纠偏平台有真空信号，无极片报警
	END_IF

//正极纠偏平台有极片，无真空信号报警
An_AlarmTon[6].IN:=NOT arrCyCtrl[arrCyNo.ElectValveName.AndeviationVacuum].Io.DIOnSwitch AND Mach_Control.An_b.An_deviationFalg 
	AND NOT Mach_Control.U.EmptyRunMode AND	arrAxisCtrl[AxiseNo.AxisName.AnCarryingUpDown].Status.Homed  
	AND arrAxisCtrl[AxiseNo.AxisName.AnCarryingUpDown].Status.fActPos<=(arrAxisPar[AxiseNo.AxisName.AnCarryingUpDown].arrTargetPoint[4]+5) 
	AND iEmptyFoldStep[1]=0 AND (DP_Step0<1000 OR DP_Step0>3100) AND NOT Mach_Control.An_b.An_VacuumErrorNG ;
	IF An_AlarmTon[6].Q  THEN
		Mach_Control.An_b.Error[6]:=TRUE;//正极纠偏平台有极片，无真空信号报警
		Mach_Control.An_b.An_VacuumErrorNG:=TRUE;//正极抛真空NG料标志
	END_IF

//正极纠偏平台连续NG
An_AlarmTon[7].IN:=Mach_Control.An_b.An_CCD_amount>=3 AND NOT Mach_Control.An_b.Error[21] AND NOT Mach_Control.U.CCD_ChosesHMI ;
	IF  An_AlarmTon[7].Q THEN
			Mach_Control.An_b.Error[21]:=TRUE;//正极纠偏平台连续NG
	END_IF	
//
IF Mach_Control.An_b.Error[24] AND CCD.AnRec.Finish.RectifyResult=3  AND rAn_AlarmRest.Q THEN
	Mach_Control.An_b.Error[24]:=FALSE;
END_IF
IF fAn_AlarmRest.Q AND Mach_Control.An_b.Error[24] AND arrAxisCtrl[AxiseNo.VirAxisName.VirMain].Status.fActPos<1  THEN	
	CCD.AnRec.Start.iPhotoDo:=1;//第二次拍照
	Mach_Control.An_b.An_CCDStart :=TRUE;//启动CCD拍照
END_IF

//正极取片报警复位
rAn_AlarmRest(CLK:=Sys_Control.btn.System_Rrestbtn , Q=> );//正极报警复位上升沿
fAn_AlarmRest(CLK:=Sys_Control.btn.System_Rrestbtn , Q=> );//正极报警复位下降沿
IF Mach_Control.U.DT_iMode=3 THEN//在手动状态下，复位报警
	
		//IF Mach_Control.An_b.Error[2] AND rAn_AlarmRest.Q THEN
				//Mach_Control.An_b.An_CarryingFalg :=FALSE;
		//END_IF
		
		IF (Mach_Control.An_b.Error[4] OR Mach_Control.An_b.Error[38]) AND rAn_AlarmRest.Q THEN
				Mach_Control.An_b.An_DPCarryingFalg:=FALSE;
		END_IF
//20240105临时屏蔽	
(*		IF Mach_Control.An_b.Error[6] AND rAn_AlarmRest.Q  THEN
				Mach_Control.An_b.An_deviationFalg :=FALSE;
		END_IF
*)		
		IF Mach_Control.An_b.Error[21] AND rAn_AlarmRest.Q  THEN
				Mach_Control.An_b.An_CCD_amount:=0;
		END_IF
																		//20240105临时屏蔽	
		IF ((Mach_Control.An_b.Error[2] AND NOT Mach_Control.An_b.An_CarryingFalg)OR Mach_Control.An_b.Error[4] OR Mach_Control.An_b.Error[38] (*OR Mach_Control.An_b.Error[6]*)) AND rAn_AlarmRest.Q  THEN
				An_StandbyStep1:=0;
				An_Step0:=0;
				An_Step1:=0;
				An_Step2:=0;
				An_Step3:=0;
		END_IF
		
		IF fAn_AlarmRest.Q AND NOT Mach_Control.An_b.Error[22]  AND NOT Mach_Control.An_b.Error[2] 
			AND NOT Mach_Control.An_b.Error[4] AND NOT Mach_Control.An_b.Error[24] 
			AND NOT Mach_Control.An_b.Error[32]  AND NOT Mach_Control.An_b.Error[34]
            AND NOT Mach_Control.An_b.Error[38] AND NOT Mach_Control.An_b.Error[39] THEN
				MEMSET(ADR(Mach_Control.An_b.Error),0,SIZEOF(Mach_Control.An_b.Error)); // 正极取片报警复位	
				//AnOverNGcount:=0;
				arrAxisCtrl[AxiseNo.AxisName.AnDTCarryingLine].Cmd.bStop:=FALSE;
		END_IF		
	
			IF AnOverNGcount>= 3 AND fAn_AlarmRest.Q THEN
		    	AnOverNGcount:=0;
		   END_IF	
		
		IF Mach_Control.An_b.An_DTqr AND Mach_Control.An_b.Error[2] THEN
			 	Mach_Control.An_b.Error[2] :=FALSE;
				Mach_Control.An_b.An_CarryingFalg :=FALSE;
		END_IF
		
		IF Mach_Control.An_b.An_DTqr AND  (Mach_Control.An_b.Error[4] OR Mach_Control.An_b.Error[38]) THEN
			 	Mach_Control.An_b.Error[4] :=FALSE;
				Mach_Control.An_b.Error[38] :=FALSE;
				Mach_Control.An_b.An_DPCarryingFalg:=FALSE;
		END_IF
		
		IF (Mach_Control.An_b.Error[7] OR An_StandbyStep0=9999) AND fAn_AlarmRest.Q THEN
				Mach_Control.An_b.Error[7] :=FALSE;
				An_StandbyStep0:=0;
		END_IF
		
		IF fAn_AlarmRest.Q THEN
				IF 9991<=An_StandbyStep1 AND An_StandbyStep1<=10000 THEN
						An_StandbyStep1:=1000;
						An_Step0:=0;
						An_Step1:=0;
						An_Step2:=0;
						An_Step3:=0;
				END_IF
		END_IF
END_IF

     An_dppy_Xzb:=arrAxisPar[AxiseNo.AxisName.AnCarryingLine].arrTargetPoint[2]+arrAxisCtrl[AxiseNo.AxisName.AnDTCarryingLine].Status.fActPos;

    IF An_Step3=30 AND NOT arrAxis[AxiseNo.AxisName.AnDTCarryingLine].Status.Coupled AND  NOT arrAxis[AxiseNo.AxisName.AnCarryingLine].Status.Coupled   AND   arrAxis[AxiseNo.VirAxisName.VirMain].Status.NotMoving 
		  AND arrAxisCtrl[AxiseNo.AxisName.AnCarryingLine].Status.Homed AND arrAxisCtrl[AxiseNo.AxisName.AnDTCarryingLine].Status.Homed AND NOT  arrAxisCtrl[AxiseNo.AxisName.AnCarryingLine].Cmd.arrbRealPoint[1]
          AND ABS((arrAxisPar[AxiseNo.AxisName.AnCarryingLine].arrTargetPoint[2]+arrAxisCtrl[AxiseNo.AxisName.AnDTCarryingLine].Status.fActPos)-arrAxisCtrl[AxiseNo.AxisName.AnCarryingLine].Status.fActPos)
            <(ABS(arrAxisPar[AxiseNo.AxisName.AnCarryingLine].arrTargetPoint[2]-arrAxisPar[AxiseNo.AxisName.AnCarryingLine].arrTargetPoint[1])+arrAxisPar[AxiseNo.AxisName.AnDTCarryingLine].arrTargetPoint[1]-20) THEN
	   Mach_Control.An_b.Error[26]:=TRUE;//正极搬运防撞软限位报警
	END_IF
	
	AnError_r(CLK:= Mach_Control.An_b.Error[26] , Q=> );
	IF AnError_r.Q THEN 
	   arrAxisCtrl[AxiseNo.AxisName.AnCarryingLine].Cmd.bStop:=TRUE;
       arrAxisCtrl[AxiseNo.AxisName.AnDTCarryingLine].Cmd.bStop :=TRUE;
	 END_IF
	 
	IF  P2M2_sysControl.btn.System_Rrestbtn THEN
			arrAxisCtrl[AxiseNo.AxisName.AnCarryingLine].Cmd.bStop:=FALSE;
			arrAxisCtrl[AxiseNo.AxisName.AnDTCarryingLine].Cmd.bStop :=FALSE;
	END_IF

	
//空叠隔膜时检查叠台升降有没有片
IF Mach_Control.U.DT_iMode=3 THEN//在手动状态下，复位报警	
		IF  Mach_Control.An_b.Error[28] AND DP_Step0=2070 AND rAn_AlarmRest.Q  THEN
				Mach_Control.An_b.An_DPCarryingFalg:=FALSE;
		END_IF
END_IF

//ccdJ拍照检测返回结果超时报警
rAnCCDStart(CLK:=Mach_Control.An_b.An_CCDStart , Q=> );
IF rAnCCDStart.Q THEN
  	 AnCCDMark:=TRUE;
END_IF
 
IF AnCCDMark AND CCD.AnRec.Finish.RectifyResult=0  AND NOT Mach_Control.U.CCD_ChosesHMI THEN
		IF NOT An_AlarmTon[12].Q THEN
			An_AlarmTon[12].IN:=TRUE;
		ELSE
			Mach_Control.An_b.Error[18] :=TRUE;//正极CCD纠偏平台检测返回结果超时
			AnCCDMark :=FALSE;
		END_IF
ELSE
		An_AlarmTon[12].IN:=FALSE;
END_IF

IF (Mach_Control.An_b.Error[18] AND Sys_Control.btn.System_Rrestbtn) OR
	   (CCD.AnRec.Finish.RectifyResult<>0 AND  AnCCDMark  AND An_AlarmTon[13].Q  ) THEN
	   AnCCDMark :=FALSE;
	   An_AlarmTon[12].IN:=FALSE;
END_IF

IF Mach_Control.U.DT_iMode=1 AND  rAnUse[4].Q THEN
 Par.stDT_date.An_sucker1_JS :=Par.stDT_date.An_sucker1_JS+1;
END_IF

IF( HMI_Hour>=7  AND HMI_Hour<9) OR (HMI_Hour>=19  AND HMI_Hour<21) THEN
      IF Par.stDT_date.An_sucker1_JS>=Par.stDT_date.An_sucker1Set THEN
	      Mach_Control.An_b.Error[42]:=TRUE;//正极送片搬运吸盘计数到达设定值
      END_IF
END_IF
IF Mach_Control.DT_b.An_sucker1_JSclear THEN
   Par.stDT_date.An_sucker1_JS:=0;
END_IF  

IF Mach_Control.U.DT_iMode=1 AND  rAnUse[5].Q THEN
 Par.stDT_date.An_sucker2_JS  :=Par.stDT_date.An_sucker2_JS +1;
END_IF

IF( HMI_Hour>=7  AND HMI_Hour<9) OR (HMI_Hour>=19  AND HMI_Hour<21) THEN
      IF Par.stDT_date.An_sucker2_JS >=Par.stDT_date.An_sucker2Set  THEN
	      Mach_Control.An_b.Error[43]:=TRUE;//正极叠台搬运吸盘计数到达设定值
      END_IF
END_IF
IF Mach_Control.DT_b.An_sucker2_JSclear THEN
   Par.stDT_date.An_sucker2_JS:=0;
END_IF  
(*
IF An_CCDNG>=10 THEN
		Mach_Control.An_b.Error[12]:=TRUE;//正极NG收纳盒满料报警
END_IF

IF Mach_Control.An_b.Error[12] AND P2M2_sysControl.btn.System_Rrestbtn THEN
		 Mach_Control.An_b.Error[12]:=FALSE;
		 An_CCDNG:=0;
END_IF

*)
END_ACTION

ACTION An_Cam:
An_Cam_ton[1](PT:=T#100MS);
An_Cam_ton[2](PT:=T#100MS);
An_Cam_ton[3](PT:=T#100MS);
An_Cam_ton[4](PT:=T#100MS);
An_Cam_ton[5](PT:=T#100MS);

(***********************************正极凸轮表创建************************************************)
(*
     fbCrectCamLeftYDLine                   :FB_CrectCamYaDaoLine ;
     fbCrectCamLeftYDUpDown             :FB_CrectCamYaDaoUpDown ;
     fbCrectCamRightYDLine                 :FB_CrectCamYaDaoLine ;
     fbCrectCamRightYDUpDown           :FB_CrectCamYaDaoUpDown ;
*)
//正极送纠偏搬运平移凸轮创建
fbAnCrectCamCarryingLine.fMoveLength:=ABS(arrAxisPar[AxiseNo.AxisName.AnCarryingLine].arrTargetPoint[1]-arrAxisPar[AxiseNo.AxisName.AnCarryingLine].arrTargetPoint[2]);
fbAnCrectCamCarryingLine(
	bCreatTable:=                fbAnCrectCamCarryingLine.bCreatTable , 
	Reset:=                          stSysState.bReset  ,  
	iTable:=                       TableNo.M_AnCarryingLine  , 
	fMoveLength:=              , 
	fMasterKeyPos:=          250 , //
	
	axisMaster:=                 arrAxis[AxiseNo.VirAxisName.VirMain] ,  
    axisSlave:=                    arrAxis[AxiseNo.AxisName.AnCarryingLine] ,  
	bCreatTableDone=> , 
	bCreatTableError=> , 
	bError=> );

fbAnCrectCamCarryingLine.bCreatTableDone;
fbAnCrectCamCarryingLine.bCreatTableError;
fbAnCrectCamCarryingLine.bError;
//正极送纠偏搬运升降取片凸轮创建
(*
fbAnCrectCamCarryingUpDown(
	bCreatTable:=fbAnCrectCamCarryingUpDown.bCreatTable, 
	Reset:=stSysState.bReset  , 
	iTable:=TableNo.M_AnCarryingUpDown , 
	fMoveLength:=arrAxisPar[AxiseNo.AxisName.AnCarryingUpDown].arrTargetPoint[2], //取片高度
	fSaveLength:=arrAxisPar[AxiseNo.AxisName.AnCarryingUpDown].arrTargetPoint[1] , //安全高度
	fInitLength:=arrAxisPar[AxiseNo.AxisName.AnCarryingUpDown].arrTargetPoint[4],//升降轴耦合初始位
	fMasterKeyPos1:=90 , //72
	fMasterKeyPos2:=180 , //144
	fMasterKeyPos3:=229 , //198
	fMasterKeyPos4:=310 , //324
	axisSlave:=arrAxis[AxiseNo.AxisName.AnCarryingUpDown]  , 
	axisMaster:=arrAxis[AxiseNo.VirAxisName.VirMain]  , 
	bCreatTableDone=> , 
	bCreatTableError=> , 
	bError=> );
	
fbAnCrectCamCarryingUpDown.bCreatTableDone;
fbAnCrectCamCarryingUpDown.bCreatTableError;
fbAnCrectCamCarryingUpDown.bError;
*)


fbAnCrectCamUpDown_4(//无用
	bCreatTable:=fbAnCrectCamUpDown_4.bCreatTable , 
	Reset:=fbAnCrectCamUpDown_4.Reset , 
	iTable:=TableNo.M_AnCarryingUpDown  , 
	fInitLength:=arrAxisPar[AxiseNo.AxisName.AnCarryingUpDown].arrTargetPoint[2], //取片高度 
	fMoveLength:=arrAxisPar[AxiseNo.AxisName.AnCarryingUpDown].arrTargetPoint[1] , //安全高度
	fSaveLength:=arrAxisPar[AxiseNo.AxisName.AnCarryingUpDown].arrTargetPoint[4],//升降轴耦合初始位
	fMasterKeyPos1:=90 , 
	fMasterKeyPos2:=180 , 
	axisSlave:=arrAxis[AxiseNo.AxisName.AnCarryingUpDown] , 
	axisMaster:=arrAxis[AxiseNo.VirAxisName.VirMain] , 
	bCreatTableDone=> , 
	bCreatTableError=> , 
	bError=> );

fbAnCrectCamUpDown_4.bCreatTableDone;
fbAnCrectCamUpDown_4.bCreatTableError;
fbAnCrectCamUpDown_4.bError;


(**********20240528SJ***************)
arrAxisPar[AxiseNo.AxisName.AnCarryingUpDown].arrTargetPoint[10]:=8; //等待高度  参数可调
arrAxisPar[AxiseNo.AxisName.AnCarryingUpDown].arrTargetPoint[11]:=18; //安全高度  参数可调
arrAxisPar[AxiseNo.AxisName.AnCarryingUpDown].arrTargetPoint[4]:=arrAxisPar[AxiseNo.AxisName.AnCarryingUpDown].arrTargetPoint[3]-arrAxisPar[AxiseNo.AxisName.AnCarryingUpDown].arrTargetPoint[10];  //等待位置
//arrAxisPar[AxiseNo.AxisName.AnCarryingUpDown].arrTargetPoint[1]:=arrAxisPar[AxiseNo.AxisName.AnCarryingUpDown].arrTargetPoint[3]-arrAxisPar[AxiseNo.AxisName.AnCarryingUpDown].arrTargetPoint[11];  //安全位置

//正极送纠偏搬运升降放片凸轮创建
fbAnCrectCamCarryingUpDown1(  //放片
	bCreatTable:=fbAnCrectCamCarryingUpDown1.bCreatTable, 
	Reset:=stSysState.bReset  , 
	iTable:=TableNo.M_AnCarryingUpDown1 , 
	fMoveLength:=    arrAxisPar[AxiseNo.AxisName.AnCarryingUpDown].arrTargetPoint[10]            , //放片高度
	fSaveLength:=    arrAxisPar[AxiseNo.AxisName.AnCarryingUpDown].arrTargetPoint[10]-arrAxisPar[AxiseNo.AxisName.AnCarryingUpDown].arrTargetPoint[11] , //安全抬升高度
	//fInitLength:=arrAxisPar[AxiseNo.AxisName.AnCarryingUpDown].arrTargetPoint[4] ,//升降轴耦合初始位
	fMasterKeyPos1:=125 , //
	fMasterKeyPos2:=250 , //
	fMasterKeyPos3:=260 , //
	fMasterKeyPos4:=320 , //
	fMasterKeyPos5:=359 , //
	//fMasterKeyPos6:=250 , //
	fSlaveVelo:=0.25 , //
	
	axisSlave:=arrAxis[AxiseNo.AxisName.AnCarryingUpDown]  , 
	axisMaster:=arrAxis[AxiseNo.VirAxisName.VirMain]  , 
	bCreatTableDone=> , 
	bCreatTableError=> , 
	bError=> );
	
fbAnCrectCamCarryingUpDown1.bCreatTableDone;
fbAnCrectCamCarryingUpDown1.bCreatTableError;
fbAnCrectCamCarryingUpDown1.bError;


//正极送纠偏搬运升降避让凸轮创建    (**********20240528SJ***************)
fbAnCrectCamCarryingUpDown3(  //避让
	bCreatTable:=fbAnCrectCamCarryingUpDown3.bCreatTable, 
	Reset:=stSysState.bReset  , 
	iTable:=TableNo.M_AnCarryingUpDown3 , 
	//fMoveLength:=arrAxisPar[AxiseNo.AxisName.AnCarryingUpDown].arrTargetPoint[10]  , //放片高度
	fSaveLength:=  arrAxisPar[AxiseNo.AxisName.AnCarryingUpDown].arrTargetPoint[10]-arrAxisPar[AxiseNo.AxisName.AnCarryingUpDown].arrTargetPoint[11] , //安全抬升高度
	//fInitLength:=arrAxisPar[AxiseNo.AxisName.AnCarryingUpDown].arrTargetPoint[4] ,//升降轴耦合初始位
	fMasterKeyPos1:=130 , //
	fMasterKeyPos2:=260 , //
	//fMasterKeyPos3:=260 , //
	//fMasterKeyPos4:=320 , //
	//fMasterKeyPos5:=359 , //
	//fMasterKeyPos6:=250 , //
	//fSlaveVelo:=0.25 , //
	axisSlave:=arrAxis[AxiseNo.AxisName.AnCarryingUpDown]  , 
	axisMaster:=arrAxis[AxiseNo.VirAxisName.VirMain]  , 
	bCreatTableDone=> , 
	bCreatTableError=> , 
	bError=> );	
fbAnCrectCamCarryingUpDown3.bCreatTableDone;
fbAnCrectCamCarryingUpDown3.bCreatTableError;
fbAnCrectCamCarryingUpDown3.bError;



//正极送纠偏搬运旋转凸轮创建 20240509 CF
fbAnCrectCamCarryingWhirling.fMoveLength:=ABS(arrAxisPar[AxiseNo.AxisName.AnCarryingWhirling].arrTargetPoint[1]-arrAxisPar[AxiseNo.AxisName.AnCarryingWhirling].arrTargetPoint[2]);
fbAnCrectCamCarryingWhirling(
	bCreatTable:=                fbAnCrectCamCarryingWhirling.bCreatTable , 
	Reset:=                          stSysState.bReset  ,  
	iTable:=                       TableNo.M_AnCarryingWhirling  , 
	fMoveLength:=             , 
	fMasterKeyPos:=          240 , //180
	
	axisMaster:=                 arrAxis[AxiseNo.VirAxisName.VirMain] ,  
    axisSlave:=                    arrAxis[AxiseNo.AxisName.AnCarryingWhirling] ,  
	bCreatTableDone=> , 
	bCreatTableError=> , 
	bError=> );

fbAnCrectCamCarryingWhirling.bCreatTableDone;
fbAnCrectCamCarryingWhirling.bCreatTableError;
fbAnCrectCamCarryingWhirling.bError;



//正极叠片搬运平移凸轮创建
fbAnCrectCamDTCarryingLine.fMoveLength:=ABS(arrAxisPar[AxiseNo.AxisName.AnDTCarryingLine].arrTargetPoint[1]-arrAxisPar[AxiseNo.AxisName.AnDTCarryingLine].arrTargetPoint[2]);
fbAnCrectCamDTCarryingLine(
	bCreatTable:=                fbAnCrectCamDTCarryingLine.bCreatTable , 
	Reset:=                          stSysState.bReset  ,  
	iTable:=                       TableNo.M_AnDTCarryingLine  , 
	fMoveLength:=             , 
	fMasterKeyPos:=          250 , //180
	
	axisMaster:=                 arrAxis[AxiseNo.VirAxisName.VirMain] ,  
    axisSlave:=                    arrAxis[AxiseNo.AxisName.AnDTCarryingLine] ,  
	bCreatTableDone=> , 
	bCreatTableError=> , 
	bError=> );
fbAnCrectCamDTCarryingLine.bCreatTableDone;
fbAnCrectCamDTCarryingLine.bCreatTableError;
fbAnCrectCamDTCarryingLine.bError;



(**********20240528SJ***************)
arrAxisPar[AxiseNo.AxisName.AnDTCarryingUpDown].arrTargetPoint[10]:=6; //等待高度  参数可调
arrAxisPar[AxiseNo.AxisName.AnDTCarryingUpDown].arrTargetPoint[11]:=18; //抬升高度  参数可调
arrAxisPar[AxiseNo.AxisName.AnDTCarryingUpDown].arrTargetPoint[4]:=arrAxisPar[AxiseNo.AxisName.AnDTCarryingUpDown].arrTargetPoint[3]-arrAxisPar[AxiseNo.AxisName.AnDTCarryingUpDown].arrTargetPoint[10];  //等待位置    以放片位为基准
//arrAxisPar[AxiseNo.AxisName.AnDTCarryingUpDown].arrTargetPoint[1]:=arrAxisPar[AxiseNo.AxisName.AnDTCarryingUpDown].arrTargetPoint[3]-arrAxisPar[AxiseNo.AxisName.AnDTCarryingUpDown].arrTargetPoint[11];  //安全位置

//正极叠片搬运升降取片凸轮创建
fbAnCrectCamDTCarryingUpDown(//取片
	bCreatTable:=fbAnCrectCamDTCarryingUpDown.bCreatTable, 
	Reset:=stSysState.bReset  , 
	iTable:=TableNo.M_AnDTCarryingUpDown , 
	fMoveLength:=arrAxisPar[AxiseNo.AxisName.AnDTCarryingUpDown].arrTargetPoint[10]-(arrAxisPar[AxiseNo.AxisName.AnDTCarryingUpDown].arrTargetPoint[3]-arrAxisPar[AxiseNo.AxisName.AnDTCarryingUpDown].arrTargetPoint[2]) , //取片高度
	fSaveLength:=arrAxisPar[AxiseNo.AxisName.AnDTCarryingUpDown].arrTargetPoint[10]-arrAxisPar[AxiseNo.AxisName.AnDTCarryingUpDown].arrTargetPoint[11]        , //安全高度
	//fInitLength:=arrAxisPar[AxiseNo.AxisName.AnDTCarryingUpDown].arrTargetPoint[4],//升降轴耦合初始位
	fMasterKeyPos1:=125 , //
	fMasterKeyPos2:=250 , //
	fMasterKeyPos3:=260 , //
	fMasterKeyPos4:= 320, //
	fMasterKeyPos5:=359 , //
	fMasterKeyPos6:= , //
	fSlaveVelo:=0.25 , //
	axisSlave:=arrAxis[AxiseNo.AxisName.AnDTCarryingUpDown]  , 
	axisMaster:=arrAxis[AxiseNo.VirAxisName.VirMain]  , 
	bCreatTableDone=> , 
	bCreatTableError=> , 
	bError=> );
fbAnCrectCamDTCarryingUpDown.bCreatTableDone;
fbAnCrectCamDTCarryingUpDown.bCreatTableError;
fbAnCrectCamDTCarryingUpDown.bError;


//正极叠片搬运升降放片凸轮创建
fbAnCrectCamDTCarryingUpDown1(//放片
	bCreatTable:=fbAnCrectCamDTCarryingUpDown1.bCreatTable, 
	Reset:=stSysState.bReset  , 
	iTable:=TableNo.M_AnDTCarryingUpDown1 , 
	fMoveLength:=arrAxisPar[AxiseNo.AxisName.AnDTCarryingUpDown].arrTargetPoint[10] ,//放片高度 
	fSaveLength:=arrAxisPar[AxiseNo.AxisName.AnDTCarryingUpDown].arrTargetPoint[10]-arrAxisPar[AxiseNo.AxisName.AnDTCarryingUpDown].arrTargetPoint[11]  , //安全高度
	//fInitLength:=arrAxisPar[AxiseNo.AxisName.AnDTCarryingUpDown].arrTargetPoint[4],//升降轴耦合初始位
	fMasterKeyPos1:=120 , //208
	fMasterKeyPos2:=250 , //256
	fMasterKeyPos3:=260 , //256
	fMasterKeyPos4:=342 , //328
	fMasterKeyPos5:=359 , //328
	fSlaveVelo:=0.25 , //
	axisSlave:=arrAxis[AxiseNo.AxisName.AnDTCarryingUpDown]  , 
	axisMaster:=arrAxis[AxiseNo.VirAxisName.VirMain]  , 
	bCreatTableDone=> , 
	bCreatTableError=> , 
	bError=> );
	
fbAnCrectCamDTCarryingUpDown1.bCreatTableDone;
fbAnCrectCamDTCarryingUpDown1.bCreatTableError;
fbAnCrectCamDTCarryingUpDown1.bError;

//正极叠片搬运升降避让凸轮创建
fbAnCrectCamDTCarryingUpDown3(//放片
	bCreatTable:=fbAnCrectCamDTCarryingUpDown3.bCreatTable, 
	Reset:=stSysState.bReset  , 
	iTable:=TableNo.M_AnDTCarryingUpDown3 , 
	//fMoveLength:=arrAxisPar[AxiseNo.AxisName.AnDTCarryingUpDown].arrTargetPoint[10] ,//放片高度 
	fSaveLength:=arrAxisPar[AxiseNo.AxisName.AnDTCarryingUpDown].arrTargetPoint[10]-arrAxisPar[AxiseNo.AxisName.AnDTCarryingUpDown].arrTargetPoint[11]  , //安全高度
	//fInitLength:=arrAxisPar[AxiseNo.AxisName.AnDTCarryingUpDown].arrTargetPoint[4],//升降轴耦合初始位
	fMasterKeyPos1:=130 , //208
	fMasterKeyPos2:=260 , //256
	//fMasterKeyPos3:=260 , //256
	//fMasterKeyPos4:=342 , //328
//	fMasterKeyPos5:=359 , //328
//	fSlaveVelo:=0.25 , //
	axisSlave:=arrAxis[AxiseNo.AxisName.AnDTCarryingUpDown]  , 
	axisMaster:=arrAxis[AxiseNo.VirAxisName.VirMain]  , 
	bCreatTableDone=> , 
	bCreatTableError=> , 
	bError=> );
	
fbAnCrectCamDTCarryingUpDown3.bCreatTableDone;
fbAnCrectCamDTCarryingUpDown3.bCreatTableError;
fbAnCrectCamDTCarryingUpDown3.bError;









An_CamTON(IN:= , PT:=T#0.5S , Q=> , ET=> );
IF Mach_Control.U.DT_iMode=3 OR Mach_Control.U.DT_iMode=0 THEN//在手动状态下
				//在触摸屏上创建正极取片凸轮
				//rAnCreate_TRIG(CLK:=Mach_Control.An_b.CreateCamStart , Q=> );
								rAnCreate_TRIG(CLK:=(Mach_Control.An_b.CreateCamStart 
									AND	NOT arrAxisCtrl[AxiseNo.AxisName.AnCarryingLine].Status.Coupled
									AND	NOT arrAxisCtrl[AxiseNo.AxisName.AnCarryingUpDown].Status.Coupled
									AND	NOT arrAxisCtrl[AxiseNo.AxisName.AnDTCarryingLine].Status.Coupled
									AND	NOT arrAxisCtrl[AxiseNo.AxisName.AnDTCarryingUpDown].Status.Coupled) , Q=> );
				IF rAnCreate_TRIG.Q THEN
					An_CamTON.IN:=FALSE;
					AnCrectCamStep0:=10;
					Mach_Control.An_b.Error[0]:=FALSE;
				END_IF
END_IF				
				//正极凸轮创建自动
				CASE AnCrectCamStep0 OF
					
							10:
									IF NOT An_CamTON.Q THEN
										An_CamTON.IN:=TRUE;
									   fbAnCrectCamCarryingLine.bCreatTable:=FALSE;//正极送片搬运平移凸轮创建
									   fbAnCrectCamCarryingUpDown.bCreatTable:=FALSE;//正极送片搬运升降取片凸轮创建
									  fbAnCrectCamUpDown_4.bCreatTable:=FALSE;//正极送片搬运升降取片凸轮创建
									  fbAnCrectCamCarryingUpDown1.bCreatTable:=FALSE;//正极送片搬运升降放片凸轮创建
									  fbAnCrectCamCarryingUpDown3.bCreatTable:=FALSE;//正极送片搬运升降放片凸轮创建								  
									  fbAnCrectCamCarryingWhirling.bCreatTable:=FALSE;//正极送片搬运旋转凸轮创建
									   fbAnCrectCamDTCarryingLine.bCreatTable :=FALSE;//正极叠片搬运平移凸轮创建
									   fbAnCrectCamDTCarryingUpDown.bCreatTable:=FALSE;//正极叠片搬运升降取片凸轮创建
									   fbAnCrectCamDTCarryingUpDown1.bCreatTable:=FALSE;//正极叠片搬运升降放片凸轮创建
									   fbAnCrectCamDTCarryingUpDown3.bCreatTable:=FALSE;//正极叠片搬运升降放片凸轮创建
									   Mach_Control.An_b.CreateCamDone:=FALSE;
									ELSE
										An_CamTON.IN:=FALSE;
									   AnCrectCamStep0:=11;
									 END_IF
							
							11:
								IF  NOT An_Cam_ton[1].Q THEN
									arrAxisCtrl[AxiseNo.AxisName.AnCarryingLine].Cmd.bStop:=TRUE;
									arrAxisCtrl[AxiseNo.AxisName.AnCarryingUpDown].Cmd.bStop:=TRUE;
									arrAxisCtrl[AxiseNo.AxisName.AnDTCarryingLine].Cmd.bStop:=TRUE;
									arrAxisCtrl[AxiseNo.AxisName.AnDTCarryingUpDown].Cmd.bStop:=TRUE;
									arrAxisCtrl[AxiseNo.AxisName.AnCarryingWhirling].Cmd.bStop:=TRUE;
									An_Cam_ton[1].IN:=TRUE;
								ELSE
									An_Cam_ton[1].IN:=FALSE;
									AnCrectCamStep0:=12;
									arrAxisCtrl[AxiseNo.AxisName.AnCarryingLine].Cmd.bStop:=FALSE;
									arrAxisCtrl[AxiseNo.AxisName.AnCarryingUpDown].Cmd.bStop:=FALSE;
									arrAxisCtrl[AxiseNo.AxisName.AnDTCarryingLine].Cmd.bStop:=FALSE;
									arrAxisCtrl[AxiseNo.AxisName.AnDTCarryingUpDown].Cmd.bStop:=FALSE;
									arrAxisCtrl[AxiseNo.AxisName.AnCarryingWhirling].Cmd.bStop:=FALSE;
								END_IF

							12:
								IF  NOT An_Cam_ton[2].Q THEN
									arrAxisCtrl[AxiseNo.AxisName.AnCarryingLine].Cmd.bReset:=TRUE;	
									arrAxisCtrl[AxiseNo.AxisName.AnCarryingUpDown].Cmd.bReset:=TRUE;
									arrAxisCtrl[AxiseNo.AxisName.AnDTCarryingLine].Cmd.bReset:=TRUE;
									arrAxisCtrl[AxiseNo.AxisName.AnDTCarryingUpDown].Cmd.bReset:=TRUE;
									arrAxisCtrl[AxiseNo.AxisName.AnCarryingWhirling].Cmd.bReset:=TRUE;
									An_Cam_ton[2].IN:=TRUE;
								 ELSE
									 An_Cam_ton[2].IN:=FALSE;
									 AnCrectCamStep0:=13;
									arrAxisCtrl[AxiseNo.AxisName.AnCarryingLine].Cmd.bReset:=FALSE;	
									arrAxisCtrl[AxiseNo.AxisName.AnCarryingUpDown].Cmd.bReset:=FALSE;
									arrAxisCtrl[AxiseNo.AxisName.AnDTCarryingLine].Cmd.bReset:=FALSE;
									arrAxisCtrl[AxiseNo.AxisName.AnDTCarryingUpDown].Cmd.bReset:=FALSE;
									arrAxisCtrl[AxiseNo.AxisName.AnCarryingWhirling].Cmd.bReset:=FALSE;
								 END_IF
								 
							13:
									arrAxisCtrl[AxiseNo.AxisName.AnCarryingLine].Cmd.bEnable:=TRUE;
									arrAxisCtrl[AxiseNo.AxisName.AnCarryingUpDown].Cmd.bEnable:=TRUE;
									arrAxisCtrl[AxiseNo.AxisName.AnDTCarryingLine].Cmd.bEnable:=TRUE;
									arrAxisCtrl[AxiseNo.AxisName.AnDTCarryingUpDown].Cmd.bEnable:=TRUE;
									arrAxisCtrl[AxiseNo.AxisName.AnCarryingWhirling].Cmd.bEnable:=TRUE;
									IF arrAxisCtrl[AxiseNo.AxisName.AnCarryingLine].Status.Enabled AND arrAxisCtrl[AxiseNo.AxisName.AnCarryingUpDown].Status.Enabled AND
										arrAxisCtrl[AxiseNo.AxisName.AnDTCarryingLine].Status.Enabled AND arrAxisCtrl[AxiseNo.AxisName.AnDTCarryingUpDown].Status.Enabled
										AND arrAxisCtrl[AxiseNo.AxisName.AnCarryingWhirling].Status.Enabled THEN
										 AnCrectCamStep0:=20;
									END_IF


		   
							20://创建凸轮
									  fbAnCrectCamCarryingLine.bCreatTable:=TRUE;//正极送片搬运平移凸轮创建
									  fbAnCrectCamCarryingUpDown.bCreatTable:=TRUE;//正极送片搬运升降取片凸轮创建
									  fbAnCrectCamUpDown_4.bCreatTable:=TRUE;//正极送片搬运升降取片凸轮创建
									  
									  fbAnCrectCamCarryingUpDown1.bCreatTable:=TRUE;//正极送片搬运升降放片凸轮创建
									   fbAnCrectCamCarryingUpDown3.bCreatTable:=TRUE;//正极送片搬运升降放片凸轮创建
									  fbAnCrectCamCarryingWhirling.bCreatTable:=TRUE;//正极送片搬运旋转凸轮创建
									   fbAnCrectCamDTCarryingLine.bCreatTable :=TRUE;//正极叠片搬运平移凸轮创建
									   fbAnCrectCamDTCarryingUpDown.bCreatTable:=TRUE;//正极叠片搬运升降取片凸轮创建
									   fbAnCrectCamDTCarryingUpDown1.bCreatTable:=TRUE;//正极叠片搬运升降放片凸轮创建
									    fbAnCrectCamDTCarryingUpDown3.bCreatTable:=TRUE;//正极叠片搬运升降放片凸轮创建
									   
									   Mach_Control.An_b.CreateCamDone:=FALSE;
									   AnCrectCamStep0:=30;
							30://等待凸轮创建完成
									IF fbAnCrectCamCarryingLine.bCreatTableDone AND fbAnCrectCamUpDown_4.bCreatTableDone(*fbAnCrectCamCarryingUpDown.bCreatTableDone*) AND fbAnCrectCamCarryingUpDown1.bCreatTableDone  AND fbAnCrectCamCarryingWhirling.bCreatTableDone AND 
										fbAnCrectCamDTCarryingLine.bCreatTableDone AND fbAnCrectCamDTCarryingUpDown.bCreatTableDone AND fbAnCrectCamDTCarryingUpDown1.bCreatTableDone  AND 
                                        fbAnCrectCamCarryingUpDown3.bCreatTableDone AND  fbAnCrectCamDTCarryingUpDown3.bCreatTableDone  THEN
										Mach_Control.An_b.CreateCamDone:=TRUE;
										 AnCrectCamStep0:=6666;
										ELSE
												IF fbAnCrectCamCarryingLine.bCreatTableError OR fbAnCrectCamCarryingUpDown.bCreatTableError OR fbAnCrectCamCarryingUpDown1.bCreatTableError OR fbAnCrectCamCarryingWhirling.bCreatTableError OR 
													fbAnCrectCamCarryingLine.bCreatTableError OR fbAnCrectCamDTCarryingUpDown.bCreatTableError OR fbAnCrectCamDTCarryingUpDown1.bCreatTableError OR fbAnCrectCamUpDown_4.bCreatTableError OR 
                                                  fbAnCrectCamCarryingUpDown3.bCreatTableError OR  fbAnCrectCamDTCarryingUpDown3.bCreatTableError   THEN
													Mach_Control.An_b.Error[0]:=TRUE;//正极取片凸轮创建失败报警
													AnCrectCamStep0:=9999;
												END_IF
									END_IF
				END_CASE







(***********************************正极凸轮耦合***********************************************)
(*
      fbAnCamInCarryingLine                      :FB_CamIn ;    
      fbAnCamInCarryingUpDown               :FB_CamIn ;    
      fbAnCamInDTCarryingLine                    :FB_CamIn ;    
      fbAnCamInDTCarryingUpDown             :FB_CamIn ;     
*)
//正极送片搬运平移凸轮耦合
fbAnCamInCarryingLine.ParCamIn.SlaveScaling;
fbAnCamInCarryingLine.ParCamIn.MasterScaling:=fAnScaling;//20240508 CF
fbAnCamInCarryingLine(
	Reset:=                      stSysState.bReset  , 
	bCamInExecute:=       fbAnCamInCarryingLine.bCamInExecute, 
	iTable1:=                   TableNo.M_AnCarryingLine  , 
	iTable2:=                   , 
	iTableSel:=                 , 
	ParCamIn:= , 
  	axisMaster:=            arrAxis[AxiseNo.VirAxisName.VirMain] ,  
	axisSlave:=               arrAxis[AxiseNo.AxisName.AnCarryingLine] ,  
	bError=> , 
	bReady=> , 
	bInSync=> );

(*Mach_Control.An_b.Error[9]:=*)fbAnCamInCarryingLine.bError;
fbAnCamInCarryingLine.bReady;
fbAnCamInCarryingLine.bInSync;

//正极送片搬运升降凸轮耦合
fbAnCamInCarryingUpDown(
	Reset:=                      stSysState.bReset  , 
	bCamInExecute:=       fbAnCamInCarryingUpDown.bCamInExecute, 
	iTable1:=                   TableNo.M_AnCarryingUpDown  , 
	iTable2:=                    TableNo.M_AnCarryingUpDown1 , 
	iTable3:=                    TableNo.M_AnCarryingUpDown3 , 
	iTableSel:=                  , 
	ParCamIn:=                  , 
  	axisMaster:=            arrAxis[AxiseNo.VirAxisName.VirMain] ,  
	axisSlave:=               arrAxis[AxiseNo.AxisName.AnCarryingUpDown] ,  
	bError=> , 
	bReady=> , 
	bInSync=> );

(*Mach_Control.An_b.Error[10]:=*)fbAnCamInCarryingUpDown.bError;
fbAnCamInCarryingUpDown.bReady;
fbAnCamInCarryingUpDown.bInSync;
//正极送片搬运旋转凸轮耦合
fbAnCamInCarryingWhirling.ParCamIn.SlaveScaling;
fbAnCamInCarryingWhirling.ParCamIn.MasterScaling:=fAnScaling;//20240508 CF
fbAnCamInCarryingWhirling(
	Reset:=                      stSysState.bReset  , 
	bCamInExecute:=       fbAnCamInCarryingWhirling.bCamInExecute, 
	iTable1:=                   TableNo.M_AnCarryingWhirling  , 
	iTable2:=                    , 
	iTableSel:=                  , 
	ParCamIn:=                  , 
  	axisMaster:=            arrAxis[AxiseNo.VirAxisName.VirMain] ,  
	axisSlave:=               arrAxis[AxiseNo.AxisName.AnCarryingWhirling] ,  
	bError=> , 
	bReady=> , 
	bInSync=> );

(*Mach_Control.An_b.Error[11]:=*)fbAnCamInCarryingWhirling.bError;
fbAnCamInCarryingWhirling.bReady;
fbAnCamInCarryingWhirling.bInSync;



//正极叠片搬运平移凸轮耦合
fbAnCamInDTCarryingLine.ParCamIn.SlaveScaling;
fbAnCamInDTCarryingLine(
	Reset:=                      stSysState.bReset  , 
	bCamInExecute:=       fbAnCamInDTCarryingLine.bCamInExecute, 
	iTable1:=                   TableNo.M_AnDTCarryingLine  , 
	iTable2:=                   , 
	iTableSel:=                 , 
	ParCamIn:=                , 
  	axisMaster:=            arrAxis[AxiseNo.VirAxisName.VirMain] ,  
	axisSlave:=               arrAxis[AxiseNo.AxisName.AnDTCarryingLine] ,  
	bError=> , 
	bReady=> , 
	bInSync=> );
(*Mach_Control.An_b.Error[12]:=*)fbAnCamInDTCarryingLine.bError;
fbAnCamInDTCarryingLine.bReady;
fbAnCamInDTCarryingLine.bInSync;


//正极叠片搬运升降凸轮耦合
fbAnCamInDTCarryingUpDown(
	Reset:=                      stSysState.bReset  , 
	bCamInExecute:=       fbAnCamInDTCarryingUpDown.bCamInExecute, 
	iTable1:=                   TableNo.M_AnDTCarryingUpDown  , 
	iTable2:=                    TableNo.M_AnDTCarryingUpDown1, 
	iTable3:=                    TableNo.M_AnDTCarryingUpDown3, 
	iTableSel:=                  , 
	ParCamIn:=                  , 
  	axisMaster:=            arrAxis[AxiseNo.VirAxisName.VirMain] ,  
	axisSlave:=               arrAxis[AxiseNo.AxisName.AnDTCarryingUpDown] ,  
	bError=> , 
	bReady=> , 
	bInSync=> );

(*Mach_Control.An_b.Error[13]:=*)fbAnCamInDTCarryingUpDown.bError;
fbAnCamInDTCarryingUpDown.bReady;
fbAnCamInDTCarryingUpDown.bInSync;


IF fbAnCamInCarryingLine.bError OR fbAnCamInCarryingUpDown.bError OR fbAnCamInCarryingWhirling.bError OR fbAnCamInDTCarryingLine.bError OR fbAnCamInDTCarryingUpDown.bError THEN
		Mach_Control.An_b.Error[11]:=TRUE;//正极有凸轮耦合报警
	ELSE		
		Mach_Control.An_b.Error[11]:=FALSE;
END_IF
END_ACTION

